(* CODESYS project EAS_PLC.library
   Company: ESCARRE AUTOMATIZACION Y SERVICIOS sl
   DefaultNamespace: EAS
   Version: 1.0.2
   Placeholder: EAS
   Author: EAS
   Title: EAS PLC

Project tree, tasks and I/O mapping:
  libraries: Tc2_Standard, * (Beckhoff Automation GmbH); Tc2_System, * (Beckhoff Automation GmbH); Tc3_Module, * (Beckhoff Automation GmbH); Util, * (System)
  DUTs/
    data type TipusCurva
  GVLs/
  POUs/
    PLC/
      MC/
        AddTanks/
          function block Circulation_TK [ST]
          function block fB_Intro_TK [ST]
          function block fBWash_TK [ST]
          function fCurvePerCen [ST]
        Elements/
          function block fBCalibrationLtr [ST]
          function block fBCntLiters [ST]
          function block fBHorn [ST]
          function block fbLiterCounter_by_flow [ST]
          function block fbLitersbyLevel [ST]
          function block fbMeterCounter_by_Speed [ST]
          function block fbPulseTrain [ST]
          function block fBUp_Down [ST]
          function block fbWashing_HT [ST]
        Fill/
          function block fBTemperatureFill [ST]
        Pump/
          function block fBPumpC [ST]
          function block fBPumpSpeed [ST]
        Seam/
          function block fBSeamTime [ST]
        Temperature/
          function block fBTermo [ST]
      Utils/
        AnalogConversions/
          function Canvi_Escala [ST]
          function Conv_Temp [ST]
        BitsConversions/
          function block Bits_to_Dword [ST]
          function block Bits_to_word [ST]
          function block Dword_to_bits [ST]
          function block Word_to_bits [ST]
        Counters/
          function block Calcul_Frequencia [ST]
          function block ContadorRapid [ST]
        FreqCycle/
          function block CalcFreq [ST]
          function block TCicle [ST]
        Timers/
          function block fBPulse1s [ST]
          function block TMP [ST]
          function block TMPpausa [ST]
  VISUs/
*)

// DUTs/TipusCurva
TYPE TipusCurva :
STRUCT
	Table:ARRAY [0..10] OF point;
END_STRUCT
END_TYPE

// POUs/PLC/MC/AddTanks/Circulation_TK
FUNCTION_BLOCK Circulation_TK
(*****************************************************************
Execute the recirculation of the add tank (Mac -> tank, tank -> mac) - 01/12/2021
v1.00
****************************************************************)
VAR_INPUT
	xActvRecirc:BOOL;				// Activate the function
	xPulsFinRecirc:BOOL;			// Finish the function
	xLowLevelRecirc:BOOL;			// Add tank Low level for the recirculation
	xHighLevelRecirc:BOOL;			// Add tank high level for the recirculation
	xMinimLevel:BOOL;				// Minimum tank level for the recirculation
	dwDrainTime:DWORD;				// Add tank drain time
END_VAR
VAR_OUTPUT
	xFiRecirc:BOOL;					// Recirculate finished
	xFill:BOOL;						// Add tank fill (runback)
	xIntro:BOOL;					// Add tank introduction (transfer)
END_VAR
VAR
	PararRecirculacio: BOOL;
	PararOmplerta: BOOL;
	OmplirEnRecirculacio: BOOL;
	PararIntroducio: BOOL;
	IntroduccioEnRecirculacio: BOOL;
	srPararRecirculacio : SR;
	TempoDescubrirNivBaix: TMP;
	Reircular: BOOL;
	FiBuidatCubeta: BOOL;
	BuidarCubeta: BOOL;
	TEmpoDrenatBuidat: TMP;
	srFiBuidatCubeta : SR;
END_VAR

// *********** Fin recircula por pulsador *****************
srPararRecirculacio(SET1:=xActvRecirc AND  xPulsFinRecirc, RESET:=NOT xActvRecirc , Q1=>PararRecirculacio );

Reircular := xActvRecirc AND NOT PararRecirculacio;

OmplirEnRecirculacio := Reircular AND NOT PararOmplerta;

IntroduccioEnRecirculacio := Reircular AND NOT PararIntroducio;
// ********* Pausa la introduccion si el nivel esta bajo *****************
TempoDescubrirNivBaix(xIN:=Reircular AND xLowLevelRecirc, dwSegons:=5 , xQ=> , dwTsegons=> );
PararIntroducio := NOT TempoDescubrirNivBaix.xQ; 

PararOmplerta := Reircular AND xHighLevelRecirc;

BuidarCubeta := xActvRecirc AND PararRecirculacio;

TEmpoDrenatBuidat(xIN:=BuidarCubeta AND NOT xMinimLevel, dwSegons:=dwDrainTime , xQ=> , dwTsegons=> );

srFiBuidatCubeta(SET1:=TEmpoDrenatBuidat.xQ , RESET:=NOT xActvRecirc , Q1=>FiBuidatCubeta );
// ************ Finaliza la recirculacion ********
xFiRecirc := FiBuidatCubeta;
// ************ Introduz a la maquina **********
xIntro := (BuidarCubeta AND NOT FiBuidatCubeta) OR IntroduccioEnRecirculacio;
// ************ Retorno de bano a la cubeta ********
xFill := OmplirEnRecirculacio;

END_FUNCTION_BLOCK

// POUs/PLC/Utils/Timers/TMP
FUNCTION_BLOCK TMP
(**********************************************************
Timer in seconds with a DWORD input - 29/11/2021
V1.0
*********************************************************)
VAR_INPUT
	xIN:BOOL;			// Enable Input
	dwSegons:DWORD;		// Setpoint Time (seconds) Input
END_VAR
VAR_OUTPUT
	xQ:BOOL;					// Boolean Output
	dwTsegons:DWORD;			// Currently Time (seconds) Output
END_VAR

VAR
	TEmporitz: TON;
	Temps: TIME;
	TempsTrans: TIME;
END_VAR

Temps := REAL_TO_TIME (DWORD_TO_REAL (dwSegons)*1000);

TEmporitz(IN:=xIN , PT:=Temps , Q=>xQ , ET=>TempsTrans );

dwTsegons := REAL_TO_DWORD(TIME_TO_REAL (TempsTrans)/1000);

END_FUNCTION_BLOCK

// POUs/PLC/MC/AddTanks/fB_Intro_TK
FUNCTION_BLOCK fB_Intro_TK
VAR_INPUT
	xActvIntro: BOOL;		///Enable the function
	dwCurve: DWORD;			/// Dosing curve
	dwTime: DWORD;			/// Duration Time
	rLevel: REAL;			/// Tank Level
	xLevelMin: BOOL;		/// Tank Minimun Level
	xIniCond: BOOL;			/// Initial condicions
	xPause: BOOL;			/// Pause the function
END_VAR
VAR_OUTPUT
	xFiIntro: BOOL;			/// End of the introduction
	rQTeoric: REAL;			/// Teoric Quantity of the introduction (%)
	rQreal: REAL;			/// Real Quantity of the introduction (%)
	xPrepareIntro: BOOL;	/// Prepare an Introduction
	xDosIntro: BOOL;		/// Introduct dosing (slow)
	xTransferIntro: BOOL;	/// Introduct transfering (fast)
	dwRemainingTime: DWORD;	/// Tiempo restante Intro
END_VAR
VAR
	IniciarIntro: BOOL;
	TEmpoInici: TMPPausa;
	calculQt: CHARCURVE;
	rampatems: RAMP_REAL;
	tempsreal: REAL;
	Tempsensegons: REAL;
	IntroduccioDosificada: BOOL;
	IntroduccioDirecte: BOOL;
	TempsEnPercentatge: REAL;
	TaulaCurva: ARRAY[0..10] OF point;
	RampaTempsInt: INT;
	QteoricaINT: INT;
	ERROR: BYTE;
	entradaRampa: REAL;
	NivellInicial: REAL;
	TempsNivellinim: TMPPausa;
	FiIntroDosificada: BOOL;
	TempsNivellinimDir: TMPPausa;
	FiDirecte: BOOL;
	srFiIntro: SR;
	A: INT;
	TMP_TimeRemaining: TMPPausa;
	dwActTime: DWORD;
END_VAR

// Inicia Intro
TEmpoInici(xIN:=xActvIntro AND xIniCond , dwSegons:=2 , xQ=>IniciarIntro , dwTsegons=> );

// Verifica si es introducion directa o dosificada
IF dwTime > 0
	THEN
		IntroduccioDosificada := TRUE;
		IntroduccioDirecte := FALSE;
	ELSE
		IntroduccioDosificada := FALSE;
		IntroduccioDirecte := TRUE;
END_IF

// Calculos del tiempo
Tempsensegons := DWORD_TO_REAL(dwTime*60);

IF IniciarIntro
	THEN
		EntradaRampa := Tempsensegons;
	ELSE
		EntradaRampa := 0;	
		NivellInicial := rLevel;
END_IF

// Si es introducin dosificada calcula la rampa
IF IntroduccioDosificada
	THEN
		rampatems(
			IN:= EntradaRampa, 
			ASCEND:= 1, 
			DESCEND:= Tempsensegons, 
			TIMEBASE:= T#1S, 
			RESET:= (IniciarIntro AND xPause) , 
			OUT=> tempsreal);

		TempsEnPercentatge := (tempsreal/Tempsensegons)*100;
END_IF

RampaTempsInt := REAL_TO_INT(TempsEnPercentatge*100);

TaulaCurva :=  fCurvePerCen(Curve:=DWORD_TO_INT (dwCurve));

calculQt(
	IN:= RampaTempsInt , 
	N:=11 , 
	P:=TaulaCurva , 
	OUT=>QteoricaINT , 
	ERR=>ERROR );

// Si se ha iniciado la introducion calcula el Qreal
IF IniciarIntro AND NivellInicial > 0
	THEN
		rQreal := (rLevel/NivellInicial)*100;
END_IF

rQTeoric := (INT_TO_REAL(QteoricaINT))/100;

xPrepareIntro := IniciarIntro AND NOT xFiIntro;

IF (rQreal > rQTeoric AND IniciarIntro AND IntroduccioDosificada AND NOT xFiIntro AND IniciarIntro) 
		THEN
		xDosIntro := TRUE;
	ELSE
		xDosIntro := FALSE;
END_IF

xTransferIntro := NOT(IntroduccioDosificada) AND IniciarIntro AND NOT xFiIntro;

TempsNivellinim(xIN:=NOT(xLevelMin) , dwSegons:=60 , xQ=> , dwTsegons=> );

IF 	rQTeoric <= 0 OR 
	rQTeoric <= 0 OR 
	TempsNivellinim.xQ (* OR 
	IntroduccioDosificada OR 
	IniciarIntro OR 
	NOT xLevelMin *)
	THEN
		FiIntroDosificada := TRUE;
	ELSE
		FiIntroDosificada := FALSE;
END_IF

TempsNivellinimDir(xIN:= NOT xLevelMin , dwSegons:=3 , xQ=> , dwTsegons=> );

FiDirecte := NOT IntroduccioDosificada AND IniciarIntro AND TempsNivellinimDir.xQ;


srFiIntro(  SET1:=(FiIntroDosificada OR FiDirecte) AND xActvIntro, 
			RESET:= NOT xActvIntro , Q1=>xFiIntro);

// TIEMPO RESTANTE INTRO
TMP_TimeRemaining(
	xIN:= IniciarIntro , 
	xPausa:= xPause, 
	dwSegons:= (dwTime*60), 
	xQ=> , 
	dwTsegons=> dwActTime, 
	rTsegons=> );

dwRemainingTime:= (dwTime*60)- dwActTime;


A:=A+1;

END_FUNCTION_BLOCK

// POUs/PLC/MC/AddTanks/fCurvePerCen
FUNCTION fCurvePerCen : ARRAY [0..10] OF POINT
(*******************************************************
Aquest Bloc Carrega per HardCode els valors de les les Corves percentuals.
Al demanar una corva retorna una taula de punts per a l'introduccio
=========================================
06/09/2006= Error corva7.
********************************************************)
VAR_INPUT
	Curve:INT;			// Curve (0 - 19)
END_VAR

VAR_OUTPUT

END_VAR	

VAR
END_VAR



(*Curve 0*)
IF Curve=0 THEN
fCurvePerCen[0].X:=0;
fCurvePerCen[0].Y:=10000;
fCurvePerCen[1].X:=1000;
fCurvePerCen[1].Y:=9000;
fCurvePerCen[2].X:=2000;
fCurvePerCen[2].Y:=8000;
fCurvePerCen[3].X:=3000;
fCurvePerCen[3].Y:=7000;
fCurvePerCen[4].X:=4000;
fCurvePerCen[4].Y:=6000;
fCurvePerCen[5].X:=5000;
fCurvePerCen[5].Y:=5000;
fCurvePerCen[6].X:=6000;
fCurvePerCen[6].Y:=4000;
fCurvePerCen[7].X:=7000;
fCurvePerCen[7].Y:=3000;
fCurvePerCen[8].X:=8000;
fCurvePerCen[8].Y:=2000;
fCurvePerCen[9].X:=9000;
fCurvePerCen[9].Y:=1000;
fCurvePerCen[10].X:=10000;
fCurvePerCen[10].Y:=0;
END_IF


(*Curve 1*)
IF curve=1 THEN
	fCurvePerCen[0].X:=0;
	fCurvePerCen[0].Y:=10000;
	fCurvePerCen[1].X:=1000;
	fCurvePerCen[1].Y:=9100;
	fCurvePerCen[2].X:=2000;
	fCurvePerCen[2].Y:=8200;
	fCurvePerCen[3].X:=3000;
	fCurvePerCen[3].Y:=7300;
	fCurvePerCen[4].X:=4000;
	fCurvePerCen[4].Y:=6400;
	fCurvePerCen[5].X:=5000;
	fCurvePerCen[5].Y:=5400;
	fCurvePerCen[6].X:=6000;
	fCurvePerCen[6].Y:=4500;
	fCurvePerCen[7].X:=7000;
	fCurvePerCen[7].Y:=3500;
	fCurvePerCen[8].X:=8000;
	fCurvePerCen[8].Y:=2400;
	fCurvePerCen[9].X:=9000;
	fCurvePerCen[9].Y:=1300;
	fCurvePerCen[10].X:=10000;
	fCurvePerCen[10].Y:=0;
END_IF


(*Curve 2*)
IF curve=2 THEN
	fCurvePerCen[0].X:=0;
	fCurvePerCen[0].Y:=10000;
	fCurvePerCen[1].X:=1000;
	fCurvePerCen[1].Y:=9200;
	fCurvePerCen[2].X:=2000;
	fCurvePerCen[2].Y:=8400;
	fCurvePerCen[3].X:=3000;
	fCurvePerCen[3].Y:=7600;
	fCurvePerCen[4].X:=4000;
	fCurvePerCen[4].Y:=6700;
	fCurvePerCen[5].X:=5000;
	fCurvePerCen[5].Y:=5800;
	fCurvePerCen[6].X:=6000;
	fCurvePerCen[6].Y:=4900;
	fCurvePerCen[7].X:=7000;
	fCurvePerCen[7].Y:=3900;
	fCurvePerCen[8].X:=8000;
	fCurvePerCen[8].Y:=2800;
	fCurvePerCen[9].X:=9000;
	fCurvePerCen[9].Y:=1500;
	fCurvePerCen[10].X:=10000;
	fCurvePerCen[10].Y:=0;
END_IF

(*GVL.Curve 3*)
IF Curve=3 THEN
	fCurvePerCen[0].X:=0;
	fCurvePerCen[0].Y:=10000;
	fCurvePerCen[1].X:=1000;
	fCurvePerCen[1].Y:=9300;
	fCurvePerCen[2].X:=2000;
	fCurvePerCen[2].Y:=8500;
	fCurvePerCen[3].X:=3000;
	fCurvePerCen[3].Y:=7800;
	fCurvePerCen[4].X:=4000;
	fCurvePerCen[4].Y:=7000;
	fCurvePerCen[5].X:=5000;
	fCurvePerCen[5].Y:=6200;
	fCurvePerCen[6].X:=6000;
	fCurvePerCen[6].Y:=5300;
	fCurvePerCen[7].X:=7000;
	fCurvePerCen[7].Y:=4400;
	fCurvePerCen[8].X:=8000;
	fCurvePerCen[8].Y:=3200;
	fCurvePerCen[9].X:=9000;
	fCurvePerCen[9].Y:=1800;
	fCurvePerCen[10].X:=10000;
	fCurvePerCen[10].Y:=0;
END_IF

(*GVL.Curve 4*)
IF curve=4 THEN
	fCurvePerCen[0].X:=0;
	fCurvePerCen[0].Y:=10000;
	fCurvePerCen[1].X:=1000;
	fCurvePerCen[1].Y:=9400;
	fCurvePerCen[2].X:=2000;
	fCurvePerCen[2].Y:=8600;
	fCurvePerCen[3].X:=3000;
	fCurvePerCen[3].Y:=8100;
	fCurvePerCen[4].X:=4000;
	fCurvePerCen[4].Y:=7400;
	fCurvePerCen[5].X:=5000;
	fCurvePerCen[5].Y:=6600;
	fCurvePerCen[6].X:=6000;
	fCurvePerCen[6].Y:=5700;
	fCurvePerCen[7].X:=7000;
	fCurvePerCen[7].Y:=4900;
	fCurvePerCen[8].X:=8000;
	fCurvePerCen[8].Y:=3600;
	fCurvePerCen[9].X:=9000;
	fCurvePerCen[9].Y:=2100;
	fCurvePerCen[10].X:=10000;
	fCurvePerCen[10].Y:=0;
END_IF


(*GVL.Curve 5*)
IF curve=5 THEN
	fCurvePerCen[0].X:=0;
	fCurvePerCen[0].Y:=10000;
	fCurvePerCen[1].X:=1000;
	fCurvePerCen[1].Y:=9500;
	fCurvePerCen[2].X:=2000;
	fCurvePerCen[2].Y:=8800;
	fCurvePerCen[3].X:=3000;
	fCurvePerCen[3].Y:=8300;
	fCurvePerCen[4].X:=4000;
	fCurvePerCen[4].Y:=7600;
	fCurvePerCen[5].X:=5000;
	fCurvePerCen[5].Y:=7000;
	fCurvePerCen[6].X:=6000;
	fCurvePerCen[6].Y:=6200;
	fCurvePerCen[7].X:=7000;
	fCurvePerCen[7].Y:=5400;
	fCurvePerCen[8].X:=8000;
	fCurvePerCen[8].Y:=4000;
	fCurvePerCen[9].X:=9000;
	fCurvePerCen[9].Y:=2300;
	fCurvePerCen[10].X:=10000;
	fCurvePerCen[10].Y:=0;
END_IF


(*GVL.Curve 6*)
IF curve=6 THEN
	fCurvePerCen[0].X:=0;
	fCurvePerCen[0].Y:=10000;
	fCurvePerCen[1].X:=1000;
	fCurvePerCen[1].Y:=9500;
	fCurvePerCen[2].X:=2000;
	fCurvePerCen[2].Y:=9000;
	fCurvePerCen[3].X:=3000;
	fCurvePerCen[3].Y:=8500;
	fCurvePerCen[4].X:=4000;
	fCurvePerCen[4].Y:=8000;
	fCurvePerCen[5].X:=5000;
	fCurvePerCen[5].Y:=7400;
	fCurvePerCen[6].X:=6000;
	fCurvePerCen[6].Y:=6600;
	fCurvePerCen[7].X:=7000;
	fCurvePerCen[7].Y:=5800;
	fCurvePerCen[8].X:=8000;
	fCurvePerCen[8].Y:=4400;
	fCurvePerCen[9].X:=9000;
	fCurvePerCen[9].Y:=2600;
	fCurvePerCen[10].X:=10000;
	fCurvePerCen[10].Y:=0;
END_IF


(*GVL.Curve 7*)
IF curve=7 THEN
	fCurvePerCen[0].X:=0;
	fCurvePerCen[0].Y:=10000;
	fCurvePerCen[1].X:=1000;
	fCurvePerCen[1].Y:=9600;
	fCurvePerCen[2].X:=2000;
	fCurvePerCen[2].Y:=9200;
	fCurvePerCen[3].X:=3000;
	fCurvePerCen[3].Y:=8800;
	fCurvePerCen[4].X:=4000;
	fCurvePerCen[4].Y:=8300;
	fCurvePerCen[5].X:=5000;
	fCurvePerCen[5].Y:=7800;
	fCurvePerCen[6].X:=6000;
	fCurvePerCen[6].Y:=7100;
	fCurvePerCen[7].X:=7000;
	fCurvePerCen[7].Y:=6300;
	fCurvePerCen[8].X:=8000;
	fCurvePerCen[8].Y:=4800;
	fCurvePerCen[9].X:=9000;
	fCurvePerCen[9].Y:=2800;
	fCurvePerCen[10].X:=10000;
	fCurvePerCen[10].Y:=0;
END_IF


(*GVL.Curve 8*)
IF curve=8 THEN
	fCurvePerCen[0].X:=0;
	fCurvePerCen[0].Y:=10000;
	fCurvePerCen[1].X:=1000;
	fCurvePerCen[1].Y:=9700;
	fCurvePerCen[2].X:=2000;
	fCurvePerCen[2].Y:=9400;
	fCurvePerCen[3].X:=3000;
	fCurvePerCen[3].Y:=9100;
	fCurvePerCen[4].X:=4000;
	fCurvePerCen[4].Y:=8600;
	fCurvePerCen[5].X:=5000;
	fCurvePerCen[5].Y:=8200;
	fCurvePerCen[6].X:=6000;
	fCurvePerCen[6].Y:=7500;
	fCurvePerCen[7].X:=7000;
	fCurvePerCen[7].Y:=6700;
	fCurvePerCen[8].X:=8000;
	fCurvePerCen[8].Y:=5200;
	fCurvePerCen[9].X:=9000;
	fCurvePerCen[9].Y:=3100;
	fCurvePerCen[10].X:=10000;
	fCurvePerCen[10].Y:=0;
END_IF

(*GVL.Curve 9*)
IF curve=9 THEN
	fCurvePerCen[0].X:=0;
	fCurvePerCen[0].Y:=10000;
	fCurvePerCen[1].X:=1000;
	fCurvePerCen[1].Y:=9800;
	fCurvePerCen[2].X:=2000;
	fCurvePerCen[2].Y:=9600;
	fCurvePerCen[3].X:=3000;
	fCurvePerCen[3].Y:=9300;
	fCurvePerCen[4].X:=4000;
	fCurvePerCen[4].Y:=9000;
	fCurvePerCen[5].X:=5000;
	fCurvePerCen[5].Y:=8600;
	fCurvePerCen[6].X:=6000;
	fCurvePerCen[6].Y:=7900;
	fCurvePerCen[7].X:=7000;
	fCurvePerCen[7].Y:=7100;
	fCurvePerCen[8].X:=8000;
	fCurvePerCen[8].Y:=5600;
	fCurvePerCen[9].X:=9000;
	fCurvePerCen[9].Y:=3400;
	fCurvePerCen[10].X:=10000;
	fCurvePerCen[10].Y:=0;
END_IF 

(*GVL.Curve 10*)
IF curve=10 THEN
	fCurvePerCen[0].X:=0;
	fCurvePerCen[0].Y:=10000;
	fCurvePerCen[1].X:=1000;
	fCurvePerCen[1].Y:=9000;
	fCurvePerCen[2].X:=2000;
	fCurvePerCen[2].Y:=8000;
	fCurvePerCen[3].X:=3000;
	fCurvePerCen[3].Y:=7000;
	fCurvePerCen[4].X:=4000;
	fCurvePerCen[4].Y:=6000;
	fCurvePerCen[5].X:=5000;
	fCurvePerCen[5].Y:=5000;
	fCurvePerCen[6].X:=6000;
	fCurvePerCen[6].Y:=4000;
	fCurvePerCen[7].X:=7000;
	fCurvePerCen[7].Y:=3000;
	fCurvePerCen[8].X:=8000;
	fCurvePerCen[8].Y:=2000;
	fCurvePerCen[9].X:=9000;
	fCurvePerCen[9].Y:=1000;
	fCurvePerCen[10].X:=10000;
	fCurvePerCen[10].Y:=0;
END_IF
	
	
(*GVL.Curve 11*)
IF curve=11 THEN
	fCurvePerCen[0].X:=0;
	fCurvePerCen[0].Y:=10000;
	fCurvePerCen[1].X:=1000;
	fCurvePerCen[1].Y:=8700;
	fCurvePerCen[2].X:=2000;
	fCurvePerCen[2].Y:=7600;
	fCurvePerCen[3].X:=3000;
	fCurvePerCen[3].Y:=6500;
	fCurvePerCen[4].X:=4000;
	fCurvePerCen[4].Y:=5500;
	fCurvePerCen[5].X:=5000;
	fCurvePerCen[5].Y:=4600;
	fCurvePerCen[6].X:=6000;
	fCurvePerCen[6].Y:=3600;
	fCurvePerCen[7].X:=7000;
	fCurvePerCen[7].Y:=2700;
	fCurvePerCen[8].X:=8000;
	fCurvePerCen[8].Y:=1800;
	fCurvePerCen[9].X:=9000;
	fCurvePerCen[9].Y:=900;
	fCurvePerCen[10].X:=10000;
	fCurvePerCen[10].Y:=0;
END_IF


(*GVL.Curve 12*)
IF curve=12 THEN
	fCurvePerCen[0].X:=0;
	fCurvePerCen[0].Y:=10000;
	fCurvePerCen[1].X:=1000;
	fCurvePerCen[1].Y:=8500;
	fCurvePerCen[2].X:=2000;
	fCurvePerCen[2].Y:=7200;
	fCurvePerCen[3].X:=3000;
	fCurvePerCen[3].Y:=6100;
	fCurvePerCen[4].X:=4000;
	fCurvePerCen[4].Y:=5100;
	fCurvePerCen[5].X:=5000;
	fCurvePerCen[5].Y:=4200;
	fCurvePerCen[6].X:=6000;
	fCurvePerCen[6].Y:=3300;
	fCurvePerCen[7].X:=7000;
	fCurvePerCen[7].Y:=2400;
	fCurvePerCen[8].X:=8000;
	fCurvePerCen[8].Y:=1600;
	fCurvePerCen[9].X:=9000;
	fCurvePerCen[9].Y:=800;
	fCurvePerCen[10].X:=10000;
	fCurvePerCen[10].Y:=0;
END_IF


(*GVL.Curve 13*)
IF curve=13 THEN
	fCurvePerCen[0].X:=0;
	fCurvePerCen[0].Y:=10000;
	fCurvePerCen[1].X:=1000;
	fCurvePerCen[1].Y:=8200;
	fCurvePerCen[2].X:=2000;
	fCurvePerCen[2].Y:=6800;
	fCurvePerCen[3].X:=3000;
	fCurvePerCen[3].Y:=5600;
	fCurvePerCen[4].X:=4000;
	fCurvePerCen[4].Y:=4700;
	fCurvePerCen[5].X:=5000;
	fCurvePerCen[5].Y:=3800;
	fCurvePerCen[6].X:=6000;
	fCurvePerCen[6].Y:=3000;
	fCurvePerCen[7].X:=7000;
	fCurvePerCen[7].Y:=2200;
	fCurvePerCen[8].X:=8000;
	fCurvePerCen[8].Y:=1500;
	fCurvePerCen[9].X:=9000;
	fCurvePerCen[9].Y:=700;
	fCurvePerCen[10].X:=10000;
	fCurvePerCen[10].Y:=0;
END_IF


(*GVL.Curve 14*)
IF curve=14 THEN
	fCurvePerCen[0].X:=0;
	fCurvePerCen[0].Y:=10000;
	fCurvePerCen[1].X:=1000;
	fCurvePerCen[1].Y:=7900;
	fCurvePerCen[2].X:=2000;
	fCurvePerCen[2].Y:=6400;
	fCurvePerCen[3].X:=3000;
	fCurvePerCen[3].Y:=5100;
	fCurvePerCen[4].X:=4000;
	fCurvePerCen[4].Y:=4300;
	fCurvePerCen[5].X:=5000;
	fCurvePerCen[5].Y:=3400;
	fCurvePerCen[6].X:=6000;
	fCurvePerCen[6].Y:=2600;
	fCurvePerCen[7].X:=5000;
	fCurvePerCen[7].Y:=1900;
	fCurvePerCen[8].X:=8000;
	fCurvePerCen[8].Y:=1400;
	fCurvePerCen[9].X:=9000;
	fCurvePerCen[9].Y:=600;
	fCurvePerCen[10].X:=10000;
	fCurvePerCen[10].Y:=0;
END_IF


(*GVL.Curve 15*)
IF curve=15 THEN
	fCurvePerCen[0].X:=0;
	fCurvePerCen[0].Y:=10000;
	fCurvePerCen[1].X:=1000;
	fCurvePerCen[1].Y:=7700;
	fCurvePerCen[2].X:=2000;
	fCurvePerCen[2].Y:=6000;
	fCurvePerCen[3].X:=3000;
	fCurvePerCen[3].Y:=4600;
	fCurvePerCen[4].X:=4000;
	fCurvePerCen[4].Y:=3800;
	fCurvePerCen[5].X:=5000;
	fCurvePerCen[5].Y:=3000;
	fCurvePerCen[6].X:=6000;
	fCurvePerCen[6].Y:=2400;
	fCurvePerCen[7].X:=7000;
	fCurvePerCen[7].Y:=1700;
	fCurvePerCen[8].X:=8000;
	fCurvePerCen[8].Y:=1200;
	fCurvePerCen[9].X:=9000;
	fCurvePerCen[9].Y:=500;
	fCurvePerCen[10].X:=10000;
	fCurvePerCen[10].Y:=0;
END_IF

(*GVL.Curve 16*)
IF curve=16 THEN
	fCurvePerCen[0].X:=0;
	fCurvePerCen[0].Y:=10000;
	fCurvePerCen[1].X:=1000;
	fCurvePerCen[1].Y:=7400;
	fCurvePerCen[2].X:=2000;
	fCurvePerCen[2].Y:=5600;
	fCurvePerCen[3].X:=3000;
	fCurvePerCen[3].Y:=4200;
	fCurvePerCen[4].X:=4000;
	fCurvePerCen[4].Y:=3400;
	fCurvePerCen[5].X:=5000;
	fCurvePerCen[5].Y:=2600;
	fCurvePerCen[6].X:=6000;
	fCurvePerCen[6].Y:=2000;
	fCurvePerCen[7].X:=7000;
	fCurvePerCen[7].Y:=1500;
	fCurvePerCen[8].X:=8000;
	fCurvePerCen[8].Y:=1000;
	fCurvePerCen[9].X:=9000;
	fCurvePerCen[9].Y:=500;
	fCurvePerCen[10].X:=10000;
	fCurvePerCen[10].Y:=0;
END_IF


(*GVL.Curve 17*)
IF curve=17 THEN
	fCurvePerCen[0].X:=0;
	fCurvePerCen[0].Y:=10000;
	fCurvePerCen[1].X:=1000;
	fCurvePerCen[1].Y:=7200;
	fCurvePerCen[2].X:=2000;
	fCurvePerCen[2].Y:=5200;
	fCurvePerCen[3].X:=3000;
	fCurvePerCen[3].Y:=3700;
	fCurvePerCen[4].X:=4000;
	fCurvePerCen[4].Y:=2900;
	fCurvePerCen[5].X:=5000;
	fCurvePerCen[5].Y:=2200;
	fCurvePerCen[6].X:=6000;
	fCurvePerCen[6].Y:=1700;
	fCurvePerCen[7].X:=7000;
	fCurvePerCen[7].Y:=1200;
	fCurvePerCen[8].X:=8000;
	fCurvePerCen[8].Y:=800;
	fCurvePerCen[9].X:=9000;
	fCurvePerCen[9].Y:=400;
	fCurvePerCen[10].X:=10000;
	fCurvePerCen[10].Y:=0;
END_IF


(*GVL.Curve 18*)
IF curve=18 THEN
	fCurvePerCen[0].X:=0;
	fCurvePerCen[0].Y:=10000;
	fCurvePerCen[1].X:=1000;
	fCurvePerCen[1].Y:=6900;
	fCurvePerCen[2].X:=2000;
	fCurvePerCen[2].Y:=4800;
	fCurvePerCen[3].X:=3000;
	fCurvePerCen[3].Y:=3300;
	fCurvePerCen[4].X:=4000;
	fCurvePerCen[4].Y:=2500;
	fCurvePerCen[5].X:=5000;
	fCurvePerCen[5].Y:=1800;
	fCurvePerCen[6].X:=6000;
	fCurvePerCen[6].Y:=1400;
	fCurvePerCen[7].X:=7000;
	fCurvePerCen[7].Y:=900;
	fCurvePerCen[8].X:=8000;
	fCurvePerCen[8].Y:=600;
	fCurvePerCen[9].X:=9000;
	fCurvePerCen[9].Y:=300;
	fCurvePerCen[10].X:=10000;
	fCurvePerCen[10].Y:=0;
END_IF


(*GVL.Curve 19*)
IF curve=19 THEN
	fCurvePerCen[0].X:=0;
	fCurvePerCen[0].Y:=10000;
	fCurvePerCen[1].X:=1000;
	fCurvePerCen[1].Y:=6600;
	fCurvePerCen[2].X:=2000;
	fCurvePerCen[2].Y:=4400;
	fCurvePerCen[3].X:=3000;
	fCurvePerCen[3].Y:=2900;
	fCurvePerCen[4].X:=4000;
	fCurvePerCen[4].Y:=1900;
	fCurvePerCen[5].X:=5000;
	fCurvePerCen[5].Y:=1400;
	fCurvePerCen[6].X:=6000;
	fCurvePerCen[6].Y:=1000;
	fCurvePerCen[7].X:=7000;
	fCurvePerCen[7].Y:=700;
	fCurvePerCen[8].X:=8000;
	fCurvePerCen[8].Y:=400;
	fCurvePerCen[9].X:=9000;
	fCurvePerCen[9].Y:=200;
	fCurvePerCen[10].X:=10000;
	fCurvePerCen[10].Y:=0;
END_IF

END_FUNCTION

// POUs/PLC/Utils/Timers/TMPpausa
FUNCTION_BLOCK TMPpausa
(**********************************************************
Timer in seconds (DWORD input) and an pause Input - 29/11/2021
V1.0
*********************************************************)
VAR_INPUT
	xIN:BOOL;				// Enable Input
	xPausa:BOOL;			// Pause Input
	dwSegons:DWORD;			// Setpoint Time in seconds (DWORD)
END_VAR
VAR_OUTPUT					
	xQ:BOOL;				// Boolean Output
	dwTsegons:DWORD;		// ET time in seconds(DWORD)
	rTsegons: REAL;			// ET time in seconds(REAL)

END_VAR

VAR
	TEmporitz: TON;
	Temps: TIME;
	TempsTrans: TIME;
	Pols_fin: F_TRIG;
	reset: BOOL;
	Temps_contador: TIME;
	Temps_pausa: TIME;
	contgeActual: TIME;
END_VAR

Temps := REAL_TO_TIME (DWORD_TO_REAL (dwSegons)*1000);

Pols_fin(CLK:=xPausa , Q=>reset);

IF	xPausa 
	THEN
		contgeActual := TEmporitz.ET;
END_IF

IF xPausa AND contgeActual > T#0S
	THEN
		Temps_pausa:= contgeActual;
		TempsTrans := Temps_pausa + TempsTrans; 
END_IF

TEmps_contador := Temps-TempsTrans;

TEmporitz(IN:=xIn AND NOT xPausa AND NOT reset, PT:=TEmps_contador , Q=>xQ , ET=>contgeActual );

IF NOT xIn
	THEN
	TEmps_contador := t#0s;
	TempsTrans := t#0s;
	Temps_pausa:= t#0s;
END_IF

dwTsegons := (REAL_TO_DWORD(TIME_TO_REAL((contgeActual)+(TempsTrans)))/1000);
rTsegons := ((TIME_TO_REAL((contgeActual)+(TempsTrans)))/1000);

END_FUNCTION_BLOCK

// POUs/PLC/MC/AddTanks/fBWash_TK
FUNCTION_BLOCK fBWash_TK
VAR_INPUT
	/// Enable function input
	xStartWash: BOOL;
	/// Minimum Level Input
	xMinimLevel: BOOL;
	/// Delay to detect the low level
	dwDetectLowLevelTime: DWORD;
	/// Drain Time
	dwDrainTime: DWORD;
	/// 1st Wash Time
	dw1stWashTime: DWORD;
	/// 2nd Wash Time
	dw2ndWashTime: DWORD;
	/// 3rd Wash Time
	dw3rdWashTime: DWORD;
	/// Drain Option (0 - 3)
	DrainType: DWORD;
END_VAR
VAR_OUTPUT
	/// Function finished			
	xFinWash: BOOL;
	/// Fill the add tank output
	xWash: BOOL;
	/// Transfer add tank to machine
	xToMachine: BOOL;
	/// Drain add tank
	xToDrain: BOOL;
END_VAR
VAR
	FerTotsElsRentats: BOOL;
	NomesRentatsAMaquina: BOOL;
	NoFerRentats: BOOL;
	FiPrimerRentat: BOOL;
	PrimerRentat: BOOL;
	TempoPrimerRentat: TMPPausa;
	FiPrimerBuidat: BOOL;
	PrimerBuidat: BOOL;
	FiSegonRentat: BOOL;
	SegonRentat: BOOL;
	FiSegonBuidat: BOOL;
	SegonBuidat: BOOL;
	TempoPrimerBuidat: TMPPausa;
	TempoSegonRentat: TMPPausa;
	TempoSegonBuidat: TMPPausa;
	TempoTercerRentat: TMPPausa;
	TempoTercerBuidat: TMPPausa;
	FiTercerRentat: BOOL;
	TercerRentat: BOOL;
	FiTercerBuidat: BOOL;
	TercerBuidat: BOOL;
	TempoBuit: TON;
	ComencaArentar: BOOL;
	BuidaDelTot: BOOL;
	srComencaArentar: SR;
	srFiPrimerRentat: SR;
	srFiPrimerBuidat: SR;
	srFiSegonRentat: SR;
	srFiSegonBuidat: SR;
	srFiTercerRentat: SR;
	srFiTercerBuidat: SR;
	FiTercer: BOOL;
	D: TMPPausa;
END_VAR

// ********** Define el tipo de lavado ***********
CASE DrainType OF
	0 : FerTotsElsRentats := TRUE;
		NoFerRentats := FALSE;
		NomesRentatsAMaquina := FALSE;
	1 : FerTotsElsRentats := FALSE;
		NoFerRentats := TRUE;
		NomesRentatsAMaquina := FALSE;
	2 : FerTotsElsRentats := FALSE;
		NoFerRentats := FALSE;
		NomesRentatsAMaquina := TRUE;
	3 : FerTotsElsRentats := TRUE;
		NoFerRentats := FALSE;
		NomesRentatsAMaquina := FALSE;
END_CASE

// ************** Empeza el lavado **************
TempoBuit(IN:= xStartWash AND NOT xMinimLevel, PT:=T#2S , Q=> , ET=> );

srComencaArentar(SET1:=TempoBuit.Q , RESET:= NOT xStartWash , Q1=>ComencaArentar );

BuidaDelTot := xStartWash AND NOT ComencaArentar;

// ********** Control Primer Lavado ******************
PrimerRentat := ComencaArentar AND NOT FiPrimerRentat;

TempoPrimerRentat(
	xIN:= ComencaArentar, 
	xPausa:= , 
	dwSegons:= dw1stWashTime, 
	xQ=> , 
	dwTsegons=> , 
	rTsegons=> );

srFiPrimerRentat(SET1:=TempoPrimerRentat.XQ , RESET:= NOT xStartWash , Q1=>FiPrimerRentat );

PrimerBuidat := FiPrimerRentat AND NOT FiPrimerBuidat;

TempoPrimerBuidat(
	xIN:= PrimerBuidat AND NOT  xMinimLevel, 
	xPausa:= , 
	dwSegons:=dwDetectLowLevelTime , 
	xQ=> , 
	dwTsegons=> , 
	rTsegons=> );

srFiPrimerBuidat(SET1:=TempoPrimerBuidat.XQ , RESET:=NOT xStartWash  , Q1=>FiPrimerBuidat );



// ********** Control Segun Lavado ***************** 
SegonRentat := FiPrimerBuidat AND NOT FiSegonRentat;

TempoSegonRentat(
	xIN:= SegonRentat , 
	xPausa:= , 
	dwSegons:= dw2ndWashTime, 
	xQ=> , 
	dwTsegons=> , 
	rTsegons=> );

srFiSegonRentat(SET1:=TempoSegonRentat.XQ , RESET:=NOT xStartWash  , Q1=>FiSegonRentat );

SegonBuidat := FiSegonRentat AND NOT FiSegonBuidat;

TempoSegonBuidat(
	xIN:= SegonBuidat AND NOT xMinimLevel, 
	xPausa:= , 
	dwSegons:= dwDetectLowLevelTime, 
	xQ=> , 
	dwTsegons=> , 
	rTsegons=> );

srFiSegonBuidat(SET1:=TempoSegonBuidat.XQ , RESET:=NOT xStartWash  , Q1=>FiSegonBuidat );

// ********** Control Tercer Lavado ***************** 
TercerRentat := FiSegonBuidat AND NOT FiTercerRentat;

TempoTercerRentat(
	xIN:= TercerRentat, 
	xPausa:= , 
	dwSegons:= dw3rdWashTime, 
	xQ=> , 
	dwTsegons=> , 
	rTsegons=> );

srFiTercerRentat(SET1:=TempoTercerRentat.XQ , RESET:=NOT xStartWash  , Q1=>FiTercerRentat );

TercerBuidat := FiTercerRentat AND NOT FiTercerBuidat;

TempoTercerBuidat(
	xIN:= TercerBuidat AND NOT xMinimLevel, 
	xPausa:= , 
	dwSegons:= dwDrainTime, 
	xQ=> , 
	dwTsegons=> , 
	rTsegons=> );

srFiTercerBuidat(SET1:=TempoTercerBuidat.XQ , RESET:=NOT xStartWash  , Q1=>FiTercerBuidat);

// ************* Finaliza los lavados ****************
xFinWash := xStartWash AND ((FerTotsElsRentats AND FiTercerBuidat) OR 
							(NomesRentatsAMaquina AND FiSegonBuidat) OR 
							NoFerRentats);// AND FiPrimerBuidat));

IF xFinWash THEN
	xStartWash := FALSE;
END_IF

// ************** Activa salidas *************
xWash	:= xStartWash AND (PrimerRentat OR SegonRentat OR TercerRentat);

xToMachine := NOT xFinWash AND (PrimerBuidat OR SegonBuidat OR BuidaDelTot);

xToDrain := NOT xFinWash AND TercerBuidat;

END_FUNCTION_BLOCK

// POUs/PLC/MC/Elements/fBCalibrationLtr
FUNCTION_BLOCK fBCalibrationLtr
//*************************************************************************************
// Con esta funcion se calibra el factor de forma de 
//
//
//*************************************************************************************

VAR_INPUT
	xStart: BOOL;		///Inicio Calibracion
	xSegOK: BOOL;		///Seguridades de máquina ok (Temp. block o Presión Min.)
	wNivel: WORD;		///Analógica de nivel debe estar ser entre 0 y 100%
	rLitros: REAL;		///Valor de litros en real
	xPause: BOOL;		///Pausa la calibracion cerrando el agua de entrada
END_VAR
VAR_OUTPUT
	N00: WORD;
	N10: WORD;
	N20: WORD;
	N30: WORD;
	N40: WORD;
	N50: WORD;
	N60: WORD;
	N70: WORD;
	N80: WORD;
	N90: WORD;
	N100: WORD;

	xPolsResetCntLitros: BOOL; 	///Usarlo para resetear el cuentalitros al inicio
	xLlenado: BOOL;				///Salida de llenado de maquina
	xAlMacNoVacia: BOOL;		///Alarma maquina no vacia al inicio.
	xFinCalibracion: BOOL;		///Pulso Fin Calibracion 2 seg
	rLitrosNivel: REAL;			///Litros extraidos del nivel
END_VAR

VAR
	xAMcNoVacia: BOOL;
	xInicioCalibracion: BOOL;
	RS_InicioCalibracion: RS;
	TON_FinCal: TON;
	TP_ResetCuentalitros: TP;
	TP_FinCalibracion: TP;
END_VAR


//Verificar que nivel es 0 antes de calibrar
xAMcNoVacia:= xStart AND NOT (xInicioCalibracion) AND (wNivel>=1);

// Inicio Calibracion
RS_InicioCalibracion(SET:= xStart AND (wNivel<=1), RESET1:= NOT (xStart)OR TON_FinCal.Q, Q1=> );
xInicioCalibracion:= RS_InicioCalibracion.Q1;

// Pulso al inicio para resetear el cuentalitros
TP_ResetCuentalitros(IN:= xInicioCalibracion, PT:= T#1S, Q=> , ET=> );
xPolsResetCntLitros:=TP_ResetCuentalitros.Q;

//Resetear los valores anteriores al iniciar Calibrado
IF xPolsResetCntLitros
	THEN
	N00 := 0;
	N10 := 0;
	N20 := 0;
	N30 := 0;
	N40 := 0;
	N50 := 0;
	N60 := 0;
	N70 := 0;
	N80 := 0;
	N90 := 0;
	N100 := 0;
END_IF

//Calibracion de la máquina
IF xInicioCalibracion THEN
	CASE wNivel OF
					
		0:	
			N00 := REAL_TO_WORD (rLitros);
		10:	
			N10 := REAL_TO_WORD (rLitros);
		20:	
			N20 := REAL_TO_WORD (rLitros);
		30:	
			N30 := REAL_TO_WORD (rLitros);
		40:	
			N40 := REAL_TO_WORD (rLitros);
		50:	
			N50 := REAL_TO_WORD (rLitros);
		60:	
			N60 := REAL_TO_WORD (rLitros);
		70:	
			N70 := REAL_TO_WORD (rLitros);
		80:	
			N80 := REAL_TO_WORD (rLitros);	
		90:	
			N90 := REAL_TO_WORD (rLitros);
		100:	
			N100 := REAL_TO_WORD (rLitros);	
	END_CASE
END_IF

/// Activar salida de llenado
xLlenado:= xInicioCalibracion AND (wNivel<100) AND NOT xPause ;

// Fin Calibracion
TP_FinCalibracion(IN:= xStart AND xInicioCalibracion AND (wNivel>=100) , PT:= T#1S, Q=> , ET=> );
xFinCalibracion:= TP_FinCalibracion.Q;

END_FUNCTION_BLOCK

// POUs/PLC/MC/Elements/fBCntLiters
FUNCTION_BLOCK fBCntLiters
VAR_INPUT
	xActv: BOOL;		/// Activate the counter
	xReset: BOOL;		/// Reset the liters value
	rInLiters: REAL;	/// Liters Input
END_VAR
VAR_OUTPUT
	rLiters: REAL;	/// Actual value 
END_VAR
VAR
	pResetLitros: R_TRIG;
	pInicio: R_TRIG;
	LitrosAcum: REAL;
END_VAR
VAR RETAIN
	/// Litros acumulados
	LitrosAc: REAL;
	/// Litros Inicial
	LitrosIni: REAL;
END_VAR

pInicio(CLK:=xActv );
//CARGAR LITROS INICIO
IF Pinicio.Q THEN
	LitrosIni := rInLiters;
	LitrosAcum:=rLiters;
END_IF

//CALCULAR LITROS EN PERIODO ACTIVO
IF xActv THEN
	LitrosAc := rInLiters-LitrosIni;
END_IF

//cALCULO LITROS
	rLiters := LitrosAc + LitrosAcum;


//PULSO RESET
pResetLitros(CLK:=xReset );
//rESET VALORES ACUMULADOS
IF  pResetLitros.Q THEN
	LitrosAcum := 0;	
	LitrosAc := 0;
	LitrosIni := 0;
END_IF

END_FUNCTION_BLOCK

// POUs/PLC/MC/Elements/fBHorn
FUNCTION_BLOCK fBHorn
VAR_INPUT
	axAlarm: ARRAY[1..Max_Alarmes] OF BOOL;
	axHorn: ARRAY[1..Max_Alarmes] OF BOOL;
	xStopHorn: BOOL;
END_VAR
VAR_OUTPUT
	xAlarmActv: BOOL;
	xHornActv: BOOL;
END_VAR
VAR
	iPunt: INT;
	afPulseAlarm: ARRAY[1..max_Alarmes] OF R_TRIG;
	xActvHorn: BOOL;
	fRS_Horn: Rs;
END_VAR


(*Comprobar si hay alarma activa*)
iPunt:=1;
xAlarmActv:=FALSE;
WHILE xAlarmActv=FALSE AND iPunt<WORD_TO_INT(Max_Alarmes)
	DO
	IF axAlarm[iPunt]=TRUE THEN
		xAlarmActv:=TRUE;
	END_IF
	iPunt:=iPunt+1;
END_WHILE


(*Activa o Reactiva Sirena*)

(*Pulso al Activar Sirena*)
iPunt:=1;
xActvHorn:=FALSE;
WHILE iPunt<WORD_TO_INT(Max_Alarmes) AND xActvHorn=FALSE
	DO
	afPulseAlarm[iPunt](CLK:= axHorn[iPunt]);
	xActvHorn:=afPulseAlarm[iPunt].Q AND xAlarmActv;
	iPunt:=iPunt+1;
END_WHILE
(*Marcha-Paro Sirena*)
fRS_Horn(SET:= xActvHorn, RESET1:=xStopHorn OR NOT(xAlarmActv));
xHornActv:=fRS_Horn.Q1;

END_FUNCTION_BLOCK

// POUs/PLC/MC/Elements/fbLiterCounter_by_flow
FUNCTION_BLOCK fbLiterCounter_by_flow
(*************************************************************
Convert a flow input into liters - 01/12/2021
V1.00
*************************************************************)
VAR_INPUT
	xActive : BOOL;			// Active the function
	rFlow :   REAL;			// Flow Input (l/min)
END_VAR
VAR_OUTPUT
	rLiters :   REAL;		// Liter output (REAL)
	dwLiters : 	DWORD;		//	Liter output (DDWORD)
END_VAR
VAR
	LitersSum : REAL;
	Periodecicle:Tcicle;
	ov: BOOL;
	INTEG: INTEGRAL;	
END_VAR


INTEG(
	IN:=rFlow , 
	TM:=10 , 
	RESET:=ov OR NOT xActive , 
	OUT=> LitersSum, 
	OVERFLOW=>ov );
	
rLiters := LitersSum/60;
dwLiters := REAL_TO_DWORD(LitersSum/60);

END_FUNCTION_BLOCK

// POUs/PLC/Utils/FreqCycle/TCicle
FUNCTION_BLOCK Tcicle
(**********************************************************
 - 29/11/2021
V1.00
*********************************************************)
VAR_INPUT

END_VAR
VAR_OUTPUT
	dwPeriode_Cicle:DWORD;		// Cycle Peryod
END_VAR

VAR_IN_OUT

END_VAR

VAR
	tempo: TON;
	reset: BOOL;
	t_actual: TIME;
	t_anterior: TIME;
	Periode: TIME;
END_VAR

tempo(IN:=NOT reset , PT:=T#7D , Q=>reset , ET=>t_actual );

Periode:= T_actual-T_anterior;

IF	NOT reset
	THEN
		T_anterior := T_actual;
END_IF

dwPeriode_cicle := TIME_TO_DWORD(Periode);

END_FUNCTION_BLOCK

// POUs/PLC/MC/Elements/fbLitersbyLevel
FUNCTION_BLOCK fbLitersbyLevel
(**********************************************
Convert an Level input into Liters - 01/12/2021
V1.00
***********************************************)
VAR_INPUT
	rLevel:REAL;
	dwN0:DWORD;
	dwN10:DWORD;
	dwN20:DWORD;
	dwN30:DWORD;
	dwN40:DWORD;
	dwN50:DWORD;
	dwN60:DWORD;
	dwN70:DWORD;
	dwN80:DWORD;
	dwN90:DWORD;
	dwN100:DWORD;
END_VAR
VAR_OUTPUT
	rLiters:REAL;
END_VAR
VAR
	iLiters:INT;
	LitrosMaq: CHARCURVE;
	litrosNivell:ARRAY[0..10]OF point;
END_VAR


litrosNivell[0].X := 0;
litrosNivell[0].Y := DWORD_TO_INT(dwN0);
litrosNivell[1].X := 100;
litrosNivell[1].Y := DWORD_TO_INT(dwN10);
litrosNivell[2].X := 200;
litrosNivell[2].Y := DWORD_TO_INT(dwN20);
litrosNivell[3].X := 300; 
litrosNivell[3].Y := DWORD_TO_INT(dwN30);
litrosNivell[4].X := 400;
litrosNivell[4].Y := DWORD_TO_INT(dwN40);
litrosNivell[5].X := 500;
litrosNivell[5].Y := DWORD_TO_INT(dwN50);
litrosNivell[6].X := 600;
litrosNivell[6].Y := DWORD_TO_INT(dwN60);
litrosNivell[7].X := 700;
litrosNivell[7].Y := DWORD_TO_INT(dwN70);
litrosNivell[8].X := 800;
litrosNivell[8].Y := DWORD_TO_INT(dwN80);
litrosNivell[9].X := 900;
litrosNivell[9].Y := DWORD_TO_INT(dwN90);
litrosNivell[10].X := 1000;
litrosNivell[10].Y := DWORD_TO_INT(dwN100);

LitrosMaq(
	IN:= REAL_TO_INT(rLevel*10) , 
	N:= 11, 
	P:= litrosNivell, 
	OUT=> iLiters, 
	ERR=> );

rLiters := INT_TO_REAL (iLiters);

END_FUNCTION_BLOCK

// POUs/PLC/MC/Elements/fbMeterCounter_by_Speed
FUNCTION_BLOCK fbMeterCounter_by_Speed
(*************************************************************
Convert an speed input into meters - 01/12/2021
V1.00
*************************************************************)
VAR_INPUT
	xMachineRunning:BOOL;
	xFabricPresence:BOOL;
	xReset:BOOL;
	rSpeed:REAL;
END_VAR
VAR_OUTPUT
	rMeters:REAL;
END_VAR
VAR
	ContarMetros: BOOL;
	Acumulador: ContadorRapid;
	cumulado: BOOL;
	acumulado: REAL;
	acumuladoInicial: REAL;
	acumuladofinal: REAL;
	Pulsocontador: F_TRIG;
	Acumular: BOOL;
END_VAR

ContarMetros := xMachineRunning AND xFabricPresence;

Pulsocontador(CLK:=ContarMetros , Q=>Acumular);

IF Acumular
	THEN
		acumuladoInicial := acumuladofinal;
END_IF

IF xReset
	THEN
		acumuladoInicial :=0;
		acumuladofinal :=0;
END_IF

Acumulador(bActivate:=ContarMetros AND NOT xReset , rFequency:=rSpeed , rCounter_REAL=>acumulado , dwCounter_DWORD=> );

acumuladofinal := acumulado + acumuladoInicial;

rMeters := acumuladofinal/60;

END_FUNCTION_BLOCK

// POUs/PLC/Utils/Counters/ContadorRapid
FUNCTION_BLOCK ContadorRapid
(**********************************************************
Creat an totalizer from an frequency input - 26/11/2021
V1.00
*********************************************************)
VAR_INPUT
	bActivate:BOOL;			// Start executing the function
	rFequency:REAL;			// Input Frequency
END_VAR

VAR_OUTPUT
	rCounter_REAL:REAL;
	dwCounter_DWORD:DWORD;
END_VAR

VAR
	Periodecicle:Tcicle;
	ov: BOOL;
	INTEG: INTEGRAL;
END_VAR



INTEG(
	IN:=rFequency , 
	TM:=Periodecicle.dwPeriode_Cicle , 
	RESET:= ov OR NOT bActivate , 
	OUT=> rCounter_REAL, 
	OVERFLOW=> ov);

dwCounter_DWORD := REAL_TO_DWORD(rCounter_REAL);

END_FUNCTION_BLOCK

// POUs/PLC/MC/Elements/fbPulseTrain
FUNCTION_BLOCK fbPulseTrain
(******************************************************
Generate a Pulse Train based on a % input - 12/01/2024
V1.02
*******************************************************)
VAR_INPUT
	rPorcentatge: REAL;		/// Percentual Input (0-100%)
	rPeriode_seg: REAL;		/// Period Input (sec)
	rPols_min_ms: REAL;		/// Minimum duration of the pulse output (ms)
END_VAR
VAR_OUTPUT
	xT_Pulsos: BOOL;		/// Pulse Output
END_VAR
VAR
	PararTren: BOOL;
	SegonsOFFtime: TIME;
	SegonsONtime: TIME;
	SegonsONreal: REAL;
	SegonsOFFreal: REAL;
	AperturaPulso: REAL;
	SegonsCicles: REAL;
	Tiemposinsenal: TMP;
	tempsmin: TIME;
	toff: TON;
	TON: TON;
	PulsMin: BOOL;
	TPulsMin: TP;
END_VAR

AperturaPulso := rPorcentatge;
SegonsCicles := rPeriode_seg;

SegonsONreal := (SegonsCicles*AperturaPulso)/100;

//no fer pols mes petit de pols minim en ON
IF SegonsONreal< (rPols_min_ms/1000)
	THEN
	SegonsONreal:=0;
END_IF
//no fer pols mes petit de pols minim en ON
IF SegonsONreal> SegonsCicles-(rPols_min_ms/1000)
	THEN
	SegonsONreal:=SegonsCicles;
END_IF

//CAlcular  temps OFF
SegonsOFFreal := SegonsCicles-SegonsONreal;

SegonsONtime := REAL_TO_TIME(SegonsONreal*1000);
SegonsOFFtime := REAL_TO_TIME(SegonsOFFreal*1000);


// Generador de pulsos
toff(IN:= NOT ton.Q, PT:=SegonsOFFtime , Q=> , ET=> );
ton(IN:= toff.Q, PT:=SegonsONtime , Q=> , ET=> );


xT_Pulsos := (toff.Q AND NOT PararTren) ;

END_FUNCTION_BLOCK

// POUs/PLC/MC/Elements/fBUp_Down
FUNCTION_BLOCK fBUp_Down
VAR_INPUT
	///Pulsador Subir 
	xUP: BOOL;
	///Pulsador Bajar 
	xDOWN: BOOL;
	///Velocidad para subir o bajar velocidad =100
	iFactor: INT := 100;
	rLimInf: REAL := 0;
	rLimSup: REAL := 100;
END_VAR
VAR_IN_OUT
	///Variable 
	SP: REAL;
END_VAR
VAR
	b_BaseTime: Blink;
	p_BaseTime: R_trig;
	xPulPulsado: BOOL;
	t2seg: Ton;
	t5seg: Ton;
	rFact: REAL;
	temps1: TIME := TIME#2s0ms;
	temps2: TIME := TIME#5s0ms;
	rFact1: REAL := 2.0;
	rFact2: REAL := 4;
END_VAR


(*Generar Base de tiempo par las subidad o bajadas*)
b_BaseTime(ENABLE:=TRUE , TIMELOW:=T#100MS , TIMEHIGH:=T#100MS , OUT=> );
p_BaseTime(CLK:=b_BaseTime.OUT );

(*Calcular Constante de subir o bajar *)
xPulPulsado:= xUP OR xDown;
t2seg(IN:=xPulPulsado , PT:=temps1  );
t5seg(IN:=xPulPulsado , PT:=temps2  );

IF NOT(t2seg.Q)
	THEN
	rFact:=INT_TO_REAL(iFactor)/100.0;
	ELSIF t2seg.Q AND NOT(t5seg.Q)
		THEN
		rFact:=INT_TO_REAL(iFactor)*rFact1/100.0;
		ELSIF t5seg.Q
			THEN
				rFact:=INT_TO_REAL(iFactor)*rFact2/100.0;
END_IF


(*Subir consigna*)
IF xUP AND p_BaseTime.Q
	THEN
	SP:=SP+rFact;
END_IF

(*Bajar consigna*)
IF xDOWN AND p_BaseTime.Q
	THEN
	SP:=SP-rFact;
END_IF

(*Limite Superior*)
IF SP>rLimSup THEN
	SP:=rLimSup;
END_IF

(*Limite Inferior*)
IF SP<rLimInf THEN
	SP:=rLimInf;
END_IF

END_FUNCTION_BLOCK

// POUs/PLC/MC/Elements/fbWashing_HT
FUNCTION_BLOCK fbWashing_HT
(**************************************************************
Execute a continuos washing in high temperature - 01/12/2021
V1.00
***************************************************************)
VAR_INPUT
	xStartDrain : BOOL;					// Enable the function
	xDirectDrain:BOOL;					// Enable direct drain input
	dwTimeFillAuxTank: DWORD;			// Time to transfer from machine to auxiliar tank
	dwTimeCloseAuxTank:DWORD;			// Time to finish the transfering to the auxiliar tank
	dwTimeDepAuxTank:DWORD;				// Time do depressurize auxiliar tank
	dwTimeDrainAunxTank:DWORD;			// Time to drain the auxiliar tank
	dwTimeCloseDrainAuxTank:DWORD;		// Time to garantee that the drain valve has closed
	xAlarmPauseWash:BOOL;				// Alarm Input to stop the function
	
END_VAR

VAR_OUTPUT
	xFillAuxTank:BOOL;					// Transfer from machuine to auxiliar tank
	xDepAuxTank:BOOL;					// depressurize auxiliar tank
	xDrainAuxTank:BOOL;					// Drain auxiliar tank
END_VAR

VAR
	ObrirBuidatRBB: BOOL;
	TempoPas1: TMP;
	TempoPas2: TMP;
	ObrirDespresuritzaRBB: BOOL;
	TempoPas3: TMP;
	ObrirOmplertaRBB: BOOL;
	TancarOmpertaRBB: BOOL;
	TancarBuidatRBB: BOOL;
	FiSequenciaRBB: BOOL;
	TempoPas4: TMP;
	TempoPas5: TMP;
	TemoDespesuritzaRBB: TMP;
	RBBsensePresio: BOOL;
	ObrirRespiraderoRBB: BOOL;
	FiBuidatRBB: BOOL;
	FiBuidatDirecte: F_TRIG;
	PolsFiBuidat: BOOL;
	TempSfINAL: TMP;
	ObrirBuidatAlBuidat: BOOL;
	srObrirOmplertaRBB :SR;
	srObrirRespiraderoRBB:SR;
	srPolsFiBuidat:SR;
	rtBuidatDirecte:F_TRIG;
	
	
END_VAR

// **************** Inicia el ciclo **************************
srObrirOmplertaRBB(SET1:= xStartDrain AND NOT srObrirOmplertaRBB.Q1 , RESET:=xAlarmPauseWash OR (FiSequenciaRBB AND ObrirOmplertaRBB) , Q1=>ObrirOmplertaRBB );


// **************** Temps por cada pas ************************
TempoPas1(xIN:=ObrirOmplertaRBB , dwSegons:=dwTimeFillAuxTank , xQ=>TancarOmpertaRBB , dwTsegons=> );

TempoPas2(xIN:=TancarOmpertaRBB , dwSegons:=dwTimeCloseAuxTank , xQ=>ObrirDespresuritzaRBB , dwTsegons=> );

TempoPas3(xIN:=ObrirDespresuritzaRBB , dwSegons:=dwTimeDepAuxTank , xQ=>ObrirBuidatRBB , dwTsegons=> );

TempoPas4(xIN:=ObrirBuidatRBB , dwSegons:=dwTimeDrainAunxTank , xQ=>TancarBuidatRBB , dwTsegons=> );

TempoPas5(xIN:=TancarBuidatRBB , dwSegons:=dwTimeCloseDrainAuxTank , xQ=>FiSequenciaRBB , dwTsegons=> );


srObrirRespiraderoRBB(SET1:=xDirectDrain AND NOT srObrirRespiraderoRBB.Q1, RESET:=xAlarmPauseWash OR (FiBuidatRBB AND ObrirRespiraderoRBB) , Q1=>ObrirRespiraderoRBB );

TemoDespesuritzaRBB(xIN:=ObrirRespiraderoRBB , dwSegons:=dwTimeDepAuxTank , xQ=>RBBsensePresio , dwTsegons=> );

rtBuidatDirecte(CLK:=xDirectDrain , Q=> );
srPolsFiBuidat(SET1:=rtBuidatDirecte.Q , RESET:=FiBuidatRBB , Q1=>PolsFiBuidat );

TempSfINAL(xIN:=PolsFiBuidat , dwSegons:=5 , xQ=>FiBuidatRBB , dwTsegons=> );

ObrirBuidatAlBuidat := xDirectDrain AND NOT FiBuidatRBB;

///*************************** Activa salidas ******************************
xFillAuxTank := (ObrirOmplertaRBB AND NOT TancarOmpertaRBB AND NOT xAlarmPauseWash) OR (xDirectDrain AND RBBsensePresio);

xDepAuxTank := (ObrirDespresuritzaRBB AND NOT TancarBuidatRBB AND NOT xAlarmPauseWash) OR xDirectDrain;

xDrainAuxTank := (ObrirBuidatRBB AND NOT TancarBuidatRBB AND NOT xAlarmPauseWash) OR ObrirBuidatAlBuidat;

END_FUNCTION_BLOCK

// POUs/PLC/MC/Fill/fBTemperatureFill
FUNCTION_BLOCK fBTemperatureFill
VAR_INPUT
	///Enable the temperature control
	xActiv: BOOL;
	/// Temperature SetPoint
	rTempSP: REAL;
	/// Real Temperature 
	rTempPV: REAL;
	/// Superior DeadBand 
	rDBHigh: REAL;
	/// Inferior DeadBand 
	rDBLow: REAL;
	///	Maximum time for adjust the temperature
	timMaxTime: TIME;
	///	Maximum time configure (1 - Open just cold water, 0 - Open cold and hot water, 2 - Activate Alarm)
	dwConfigMaxTime: DWORD;
	/// Minimum level input
	xLevel: BOOL;
	/// Level Configure (0 - Disable, 1 - Starts filing with CW and HW, 2 - Starts filing with CW, 3 - Starts filing with HW) 
	dwConfigLevel: DWORD;
	/// Time delay for start adjusting the teperature.
	timControl: TIME;
END_VAR
VAR_OUTPUT
	/// Cold Water Output
	xCWater: BOOL;
	/// Hot Water Output
	xHWater: BOOL;
	/// Maximum time alarm Output
	xAlarmMaxTime: BOOL;
END_VAR
VAR
	TempIni: TON;
	MaxTemp: TON;
	/// Temperatura mínima SP-DBmin	
	TemperMin: REAL;
	/// Temperatura mínima SP+DBmax
	TemperMax: REAL;
	CtrlNivel: BOOL;
	xNivOK: BOOL;
	xRegOutDB: BOOL;
END_VAR


//Delay para empezar la regulacion
TempIni(IN:=xActiv, PT:=timControl , Q=> , ET=> );

//Esperar nivel minimo si es necesario
IF dwConfigLevel > 0
	THEN
		xNivOK := xLevel;
	ELSE
		xNivOK := 1;
END_IF

//Margenes de la banda muerta de regulacion			
TemperMax := rTempSP + rDBHigh;
TemperMin := rTempSP - rDBLow;
//Temperatura Fuera banda muerta
xRegOutDB:=  ((rTempPV < TemperMin) OR (rTempPV > TemperMax));

//Tiempo maximo de regulacion
MaxTemp(	IN:=	TempIni.Q AND 						//inicia reguñacion
					xRegOutDB AND 						//Temperatura fuera banda muerta
					xNivOK  , 							//Esperar si es necesario el nivel 
			PT:=	timMaxTime ,						//tiempo maximo de regulacion 
			Q=>		xAlarmMaxTime );					//Alarma tiempo maxioms reg

			

IF xActiv
	THEN
		//Abrir 2 aguas
		IF (xRegOutDB AND (NOT MaxTemp.Q)) OR      //temp fuera banda muerta
			(MaxTemp.Q AND (dwConfigMaxTime = 0) AND (dwConfigMaxTime <> 2)) OR 
			NOT(TempIni.Q) OR 
			(dwConfigLevel = 1 AND NOT xLevel) 
			THEN
				xCWater :=TRUE;
				xHWater :=TRUE;
		END_IF	
		IF 	rTempPV > TemperMax AND 
			NOT(MaxTemp.Q) AND 
			(	TempIni.Q OR 
				(MaxTemp.Q AND dwConfigMaxTime = 1 AND dwConfigMaxTime <> 2) OR 
				(dwConfigLevel = 3 AND NOT xLevel)
			)
			THEN			
				xCWater :=TRUE;
				xHWater :=FALSE;			
		END_IF 
		IF rTempPV < TemperMin AND 
		NOT(MaxTemp.Q) AND 
		(	TempIni.Q OR 
			(dwConfigLevel = 2 AND NOT xLevel)
		)
			THEN			
				xCWater :=FALSE;
				xHWater :=TRUE;			
		END_IF
		IF MaxTemp.Q AND dwConfigMaxTime = 2
			THEN
				xCWater :=FALSE;
				xHWater :=FALSE;
		END_IF
	 ELSE
		xCWater :=FALSE;
		xHWater :=FALSE;			
END_IF

END_FUNCTION_BLOCK

// POUs/PLC/MC/Pump/fBPumpC
FUNCTION_BLOCK fBPumpC
VAR_INPUT
	///Pulsador de marcha
	fP_Run: BOOL;
	///Pulsador de paro
	fP_Stop: BOOL;
	///Pulsador de continua programa
	xP_ContProg: BOOL;
	///Nivel Seguridad Bomba
	xLvlSeg: BOOL;
	///Condiciones Seguridad arranque Bomba
	xSeg: BOOL;
	///Condiciones arrancar Bomba
	xConditionRun: BOOL;
	/// Condiciones paran bomba
	xConditionStop: BOOL;
	///1:manual  2: auto
	iAutoMan: INT;
END_VAR
VAR_OUTPUT
	Run: BOOL;
END_VAR
VAR
	xExistePulParo: BOOL;
	RT_PasoAuto: R_trig;
	xRunForPul: BOOL;
	RT_Run: R_trig;
	RT_Stop: R_trig;
	xStopForPul: BOOL;
	xArrancar: BOOL;
	xRunContProg: BOOL;
	tContProg: Ton;
	xParar: BOOL;
	RS_PUMP: Rs;
	a: INT;
	FTParoPorNoMarcha: F_TRIG;
	xParoPorNoMarcha: BOOL;
	TON_MarchaBomba: TON;
END_VAR

a:=a+1;

(*-------------------------------------------*)
(****** Condiciones de Inicio******)
//Con pulsación de 1 segundo funciona como pulsador de marcha
//Con pulsación de más de 1 segundo funciona como barra (selector)*) 

(*-----Gestion Pulsadores-----*)

(*Pulso Run*)
RT_Run(CLK:=fP_run );

(*Pulso Stop*)
RT_Stop(CLK:=fP_Stop );

(*Pulso Paro por no marcha*)
TON_MarchaBomba(IN:= fP_run, PT:= T#1S, Q=> , ET=> );
FTParoPorNoMarcha(CLK:=TON_MarchaBomba.Q , );

xParoPorNoMarcha:= FTParoPorNoMarcha.Q;

(*Pul Cont Prog,*)
tContProg(IN:=xP_ContProg , PT:=T#5S);


(*-----Paso a Auto------*)
RT_PasoAuto(CLK:= iAutoMan=2 );


(*------------------------------------*)
(*     Marcha       *) 
(*------------------------------------*)
xArrancar:= RT_Run.Q OR  			(*Arranc pulsadors*)
			tContProg.Q OR  		(*Arranc Cont Prog*)	
			RT_PasoAuto.Q OR
			xConditionRun;
			
			
(*------------------------------------*)
(*     Paro       *) 
(*------------------------------------*)
xParar:= 	RT_Stop.Q OR 			(*Paro  por pulsadores*)
			xConditionStop OR		(*Condiciones de paro*)
			//NOT(xLvlSeg) OR			(*Falta nivel de seguridad*)
			NOT(xSeg)OR
			xParoPorNoMarcha;    (*Paro cuando salimos de marcha con barra*)
			
(*------------------------------------*)
(*     Arranque       *) 
(*------------------------------------*)
			
RS_PUMP(SET:=xArrancar , RESET1:= xParar );

Run:= 	RS_pump.Q1;

END_FUNCTION_BLOCK

// POUs/PLC/MC/Pump/fBPumpSpeed
FUNCTION_BLOCK fBPumpSpeed
VAR_INPUT
	///Bomba en marcha
	xRun: BOOL;
	///0=Man  1=Auto  
	xAutoMan: BOOL;
	///Pulsador Subir Velocidad
	xUP_Speed: BOOL;
	///Pulsador Bajar Velocidad
	xDOWN_Speed: BOOL;
	///Consigna de la funcion velocidad 0..100%
	rSP_Function: REAL;
	iFACTOR: INT := 50;
END_VAR
VAR_OUTPUT
	///Consigna velocidad 0..100%
	SP_Speed: REAL;
	///Consigna velocidad Auto 0..100%
	SP_Auto: REAL;
	///Consigna velocidad Manual 0..100%
	SP_Man: REAL;
END_VAR
VAR
	GestPul: fBUP_down;
	a: INT;
END_VAR

a:=a+1;
(*GESTION SP MANUAL*)
(*cargar valor sp auto al estar en auto*)
IF (xAutoMan) THEN
	SP_Man:=SP_Auto;
END_IF

(*GESTION SP AUTO*)
SP_Auto:=rSP_Function;


(*Gestion Pulsadores*)
GestPul(
	xUP:= 		xUP_Speed, 
	xDOWN:= 	xDOWN_Speed, 
	iFactor:= 	iFACTOR, 
	rLimInf:= 	0, 
	rLimSup:= 	100, 
	SP:= SP_Man);

(*Gestion SP*)

IF xAutoMan 
	THEN
	SP_Speed:=SP_Auto;
	ELSE
	SP_Speed:=SP_Man;		
END_IF

IF NOT(xRun) 
	THEN
	SP_Speed:=0;
END_IF

END_FUNCTION_BLOCK

// POUs/PLC/MC/Seam/fBSeamTime
FUNCTION_BLOCK fBSeamTime
VAR_INPUT
	xWinchRun: BOOL;
	xControlActv: BOOL;
	xSeamDetect: BOOL;
	iPercContol: INT;
	iTimeMax: INT;
END_VAR
VAR_OUTPUT
	xStoped: BOOL;
	xCntrlRun: BOOL;
	xNoSeam: BOOL;
	xDetectionPulse: BOOL;
	iTimeAct: INT;
	iTimeAnt1: INT;
	iTimeAnt2: INT;
	iTimeAnt3: INT;
END_VAR
VAR
	///Durada del 
	tTimePulseOut: TIME := TIME#2s0ms;
	tTimePulseMin: TIME := TIME#200ms;
	tTimerMinPulse: ton;
	pPulseSeam: r_trig;
	TTimerPulse: tp;
	tTimerSeam: ton;
	iPasesParacontrol: INT := 2;
	cContPaso: CTU;
	tTimeAlarm: REAL;
	xBloqPulso: BOOL;
	tTimeMax: TIME;
END_VAR



//Asegurar un pulso minimo par descartar rebotes
tTimerMinPulse(IN:=xSeamDetect , PT:=tTimePulseMin );
pPulseSeam(CLK:=tTimerMinPulse.Q);

//Generar Pulso de deteccion con tiempo fijo
TTimerPulse(IN:= pPulseSeam.Q, PT:=tTimePulseOut );
xDetectionPulse:= TTimerPulse.Q  ;

//Bloquear pulsos por posible rebote
xBloqPulso:= (iTimeAct<(iTimeAnt1/20));

//Acumular temps de pas al detectar pas d'iman
IF xWinchRun AND pPulseSeam.Q AND NOT(xBloqPulso)
	THEN
		iTimeAnt3:=iTimeAnt2;
		iTimeAnt2:=iTimeAnt1;
		iTimeAnt1:=iTimeAct;
END_IF

//Calculo tiempo actual
tTimerSeam(	IN:=xWinchRun AND NOT(pPulseSeam.Q) AND xControlActv, 
			PT:=T#1D );

iTimeAct:=TIME_TO_INT(tTimerSeam.ET/1000);



//Control Paso de cuerda

cContPaso(
	CU:= 		xControlActv AND pPulseSeam.Q , 
	RESET:= 	NOT(xControlActv), 
	PV:= 		INT_TO_WORD(iPasesParacontrol));
	
xCntrlRun:=cContPaso.Q;

//Tiempo maximo calculado con el porcentaje
tTimeAlarm:= (INT_TO_REAL(iTimeAnt1)*(1.0+INT_TO_REAL(iPercContol)/100.0))  ;


xStoped:= 	xCntrlRun AND				//control activo
			cContPaso.Q AND 			//La cuerda ha pasado 2 veces
			(iTimeAct >	tTimeAlarm);	//tiempo actual mayor al anterior	
			
//Alarma de FALTA IMAN (xNoSeam)			
xNoSeam:= 	xCntrlRun AND				//control activo
			xWinchRun AND 				//Torniquete en marcha
			(iTimeAct >	iTimeMax);		//tiempo actual mayor el Maximo

END_FUNCTION_BLOCK

// POUs/PLC/MC/Temperature/fBTermo
FUNCTION_BLOCK fBTermo
VAR_INPUT
	///		Activa el calcul del gradient
	TermoActv: BOOL;
	///		Lectura de la temperatura 
	TemperaturaReal: REAL;
	///		Temperatura final que es vol obtenir  
	TemperaturaFinal: REAL;
	///		Expresat en decimes de grau 
	Gradient: REAL;
	///		Temps de maneniment en minuts 
	t_Manteniment: REAL;
	///		Entrada que s'utilitza com a rellotge (1seg per regular per temps) 
	Pols: BOOL;
	///		Aquesta entrada produeix una pausa en el calcul 
	PausaExterior: BOOL;
	///		Diferencia de temperatura necesaria per parar la consigna per 
	///		esperar a la temperatura real. Definit en  graus, per defecte =2  
	GrausPerIntegracio: REAL := 2;
	///		Diferencia de graus amb les que es forzara calentar encara que la
	///		temperatura sigui superior i la consigna pasarà a ser directament 
	///		la temperatura final .definit en graus i real. per defecte =4  
	GrausForzarCal: REAL := 4;
	///		Recomença la termoregulacio agafant la temperaturaimposada 
	///		com a inicial.  S'utilitza per poder modificar el gradient en una 
	///		introducció ( fa un reset a la durada i agafa el gradient actual). 
	ReIniciarTermo: BOOL;
	///		Temps seguretat per a cambiar de calentar a refredar o al reves
	///		 per defecte =30
	TmoSegConmutacion: DWORD := 30;
	///		diferencia de teperatura per realitzar la conmutació durant 
	///		el manteniment  per defecte =5
	ConmutacioEnManteniment: REAL := 5;
	BandaProporcional: REAL;
	PartIntergral: REAL;
	PartDerivada: REAL;
	T_periode: REAL;
	SeguretatOK: BOOL;
	ObrirPurgaenRepos: BOOL;
	t_Purga: DWORD;
	///Paralel: Temperatura per iniciar el calcul de la termorregulacio 
	TemperaturaPerInici: REAL;
	NO_Reset: BOOL;
END_VAR
VAR_OUTPUT
	///		Indica que la termorregulacio esta pausada per integracio
	EnIntegracio: BOOL;
	///		Indicacio de la temperatura imposada
	TemperaturaImposada: REAL;
	///		Termoregulació per calentar, Es la ordre al regulador
	Vapor: BOOL;
	Apertura_Vapor: REAL;
	///		Termoregulació per refredar, , Es la ordre al regulador 
	AiguaRefredament: BOOL;
	Apertura_Refreda: REAL;
	///		Indicacio que la temperatura a arribat a la temperatura final 
	EnManteniment: BOOL;
	Actv_RetornAigua: BOOL;
	Actv_RetornVapor: BOOL;
	Actv_BuidatSerpenti: BOOL;
	DuradaTermo: DWORD;
	///solo informacion
	refredar: BOOL;
	///solo informacion
	calentar: BOOL;
END_VAR
VAR
	TemperaturaInicial: REAL;
	TemporIniciar: TON;
	IniciarTermo: BOOL;
	TempsEnMarxa: BOOL;
	DiferencialImposada: REAL;
	DiferenciaTemp: REAL;
	ActvManteniment: BOOL;
	TempoManteniment: TON;
	errorPID: BOOL;
	ResetPID: BOOL;
	EsperaSortida: BOOL;
	OKCalentar: TMPPausa;
	OKRefredar: TMPPausa;
	TemperaturaMaxima: REAL;
	TemperaturaMinima: REAL;
	TempsTempAlta: TON;
	PasarARefredar: BOOL;
	TempsTempBaixa: TON;
	PasarACalentar: BOOL;
	Part_Proporcional: REAL;
	PI: REAL;
	Y_min: REAL;
	Y_max: REAL;
	PID_CALENTAR: PID_fixcycle;
	polsResetMant: R_TRIG;
	ResetGrad0: BOOL;
	SortidaPID: REAL;
	tempsPurga: TMPPausa;
	TR: REAL;
	TI: REAL;
	Actv_Vapor: BOOL;
	Actv_AiguaRefredament: BOOL;
	PI_reg: REAL;
	xMan: BOOL := FALSE;
	xLim: BOOL;
	xOver: BOOL;
	IN: INT;
	DE: TMPPausa;
	D: TON;
END_VAR

(*iniciar TermoRegulación*)
TemporIniciar
	(IN:= TermoActv ,
	 PT:= T#1s ,
	 Q=> IniciarTermo ,
	 ET=> );

(*Guardar valor temperatura inicial*)
IF NOT(IniciarTermo)
	THEN
		IF TemperaturaPerInici=0
			THEN
			TemperaturaInicial:=TemperaturaReal;
			DuradaTermo:=0;
			ELSE
			TemperaturaInicial:=TemperaturaPerInici;
			DuradaTermo:=0;
		END_IF
END_IF


(*Reiniciar el calcul de la consigna de la termorregulacio*)
IF ReIniciarTermo
	THEN
		TemperaturaInicial:=TemperaturaImposada;
		DuradaTermo:=0;
END_IF


(*Termoregulacio  en integració*)
IF Calentar
	THEN
		DiferenciaTemp:=TemperaturaImposada - TemperaturaReal;
END_IF
IF Refredar
	THEN
		DiferenciaTemp:=TemperaturaReal-TemperaturaImposada;
END_IF
IF (DiferenciaTemp>GrausPerIntegracio) AND TermoActv
	THEN
		EnIntegracio:=TRUE;
	ELSE
		EnIntegracio:=FALSE;
END_IF

(*Calcul del  Temps de termoregulacio*)
TempsEnMarxa:= (IniciarTermo) AND NOT(PausaExterior) AND NOT(EnManteniment) AND NOT(EnIntegracio);
IF (TempsEnMarxa) AND (Pols)
	THEN
		DuradaTermo:=DuradaTermo+1;
END_IF

(* Mirar si calenta o refreda *)
IF TermoActv
	THEN
		IF ((TemperaturaFinal+GrausForzarCal) >= (TemperaturaInicial))
			THEN
				Calentar:= TRUE;
				Refredar:= FALSE;
		END_IF
		IF ((TemperaturaFinal+GrausForzarCal) < (TemperaturaInicial))
			THEN
				Calentar:= FALSE;
				Refredar:= TRUE;
		END_IF
	ELSE
		Calentar:= FALSE;
		Refredar:= FALSE;
END_IF

(*Calcul Tamperatura*)
IF Gradient<>0
	THEN
		DiferencialImposada:= ((Gradient * DWORD_TO_REAL(DuradaTermo)) / 600.0) ;
		IF calentar
			THEN
				TemperaturaImposada:= TemperaturaInicial+DiferencialImposada;
				IF TemperaturaImposada > TemperaturaFinal
				THEN
					TemperaturaImposada := TemperaturaFinal;
				END_IF
			ELSE
				IF refredar
					THEN
						TemperaturaImposada:= TemperaturaInicial - DiferencialImposada;
					ELSE
						TemperaturaImposada := TemperaturaReal;
				END_IF
		END_IF
	ELSE
		TemperaturaImposada := TemperaturaFinal;
END_IF
IF NOT(TermoActv)
	THEN
		TemperaturaImposada := TemperaturaReal;
END_IF


(*Calcular Si esta en manteniment*)
IF gradient<>0
	THEN
		IF ((TemperaturaImposada >= TemperaturaFinal AND Calentar) OR 
			(TemperaturaImposada <= TemperaturaFinal AND Refredar))
			THEN
				ActvManteniment:=TRUE;
				TemperaturaImposada:=TemperaturaFinal;
		END_IF
	ELSE
		IF ((TemperaturaReal >= (TemperaturaFinal-(GrausPerIntegracio) ) AND Calentar) OR (TemperaturaReal <= (TemperaturaFinal + (GrausPerIntegracio)) AND Refredar))
			THEN 
				ActvManteniment:=TRUE;
		END_IF
END_IF

IF NOT(TermoActv)
	THEN
		ActvManteniment:=FALSE;
END_IF

TempoManteniment(IN:= ActvManteniment, PT:= T#5S, Q=> , ET=> );

EnManteniment:=Tempomanteniment.Q;

(*@@@@@@@@@@@@@@@@@@@@@@@@@@@@@@@@@@@@@@@@@@@@@@@@@@@@@@@@@@@@@@@@@@@@*)


(*Si no calenta ni refreda es fa un reset del pid*)
(*Reset al entrar en manteniment*)
ResetGrad0:=((TemperaturaReal >= (TemperaturaFinal-(BandaProporcional/10.0) ) AND Calentar) OR (TemperaturaReal <= (TemperaturaFinal + (BandaProporcional/10.0)) AND Refredar));
polsResetMant(CLK:= ((gradient<>0 AND EnManteniment AND NOT(no_reset)) OR (gradient=0 AND ResetGrad0))); 			(*24/05/2013 modificat*)
IF (NOT(Calentar) AND NOT(Refredar)) OR (errorPID)  OR  (polsResetMant.Q) OR pasaraCalentar OR PasaraRefredar
	THEN
		ResetPID:=TRUE;
	ELSE
		ResetPID:=FALSE;
END_IF

(*Seguretat per activar el calentament*)

OKCalentar(
		xIN:= NOT(Refredar), 
		xPausa:= FALSE, 
		dwSegons:= TmoSegConmutacion , 
		xQ=> , 
		dwTsegons=> , 
		rTsegons=> );

OKRefredar(
		xIN:= NOT(Calentar), 
		xPausa:= FALSE, 
		dwSegons:= TmoSegConmutacion , 
		xQ=> , 
		dwTsegons=> , 
		rTsegons=> );

(*Activar Calentar o Refredar  tenint en compte el mantnment*)
(*Manteniment NO actiu*)
EsperaSortida:= (EnManteniment AND ((calentar AND okcalentar.xQ) OR (refredar AND okrefredar.xQ)));
IF NOT(EnManteniment) OR NOT EsperaSortida
	THEN
		Actv_Vapor :=Calentar AND okcalentar.xQ;
		Actv_AiguaRefredament :=Refredar AND okrefredar.xQ ;
END_IF
(*Manteniment SI actiu*)
(* Temperatures per fer les conmutacions *)
TemperaturaMaxima := TemperaturaImposada + (ConmutacioEnManteniment);
TemperaturaMinima := TemperaturaImposada - (ConmutacioEnManteniment);
(*Pasar  de calentar a refredar*)

TempsTempAlta(IN:= ((Actv_Vapor)AND(TemperaturaMaxima<TemperaturaReal)AND(EnManteniment)), 	
					PT:=T#5S , 
					Q=> PasarARefredar, ET=> );

IF PasarARefredar
	THEN
		Actv_Vapor:=FALSE;
		Actv_AiguaRefredament:=TRUE;
END_IF
(*Pasar  de refredar a calentar*)

TempsTempBaixa(IN:= ((Actv_AiguaRefredament)AND(TemperaturaMinima>TemperaturaReal)AND(EnManteniment)), 
					PT:= T#5S, 
					Q=> PasarACalentar, 
					ET=> );

IF PasarACalentar
	THEN
		Actv_Vapor:=TRUE;
		Actv_AiguaRefredament:=FALSE;
END_IF

(*Preparar valors del PID*)
(* BandaProporcional *)
IF BandaProporcional=0
	THEN
		BandaProporcional:=10.0;
END_IF
(*Calcul Part Proorcional*)
Part_Proporcional:=(1000.0/BandaProporcional);
(* Part integral*)
IF Gradient=0 AND NOT(enmanteniment)
THEN
PI:=0;
ELSE
PI:=PartIntergral;
END_IF
(*Maxim i minim *)
		Y_min:=0;
		Y_max:=100;
(*Temperatures PID*)
IF Actv_Vapor
	THEN
		TR:=TemperaturaReal;
		TI:=TemperaturaImposada;
END_IF
IF Actv_AiguaRefredament
	THEN
		TR:=300-TemperaturaReal;
		TI:=300-TemperaturaImposada;
END_IF

IF PI<=0 THEN
	PI_reg:=1E+36;
	ELSE
	PI_reg:=PI;	
	END_IF

PID_CALENTAR(
	ACTUAL:= 	TR, 
	SET_POINT:= TI, 
	KP:= 		Part_Proporcional, 
	TN:=		PI_reg , 
	TV:= 		PartDerivada, 
	Y_MANUAL:= 	0, 
	Y_OFFSET:= 	0, 
	Y_MIN:= 	Y_min, 
	Y_MAX:= 	Y_max, 
	MANUAL:= 	xMan, 
	RESET:= 	ResetPID, //Activar al cambiar el PID
	CYCLE:= 	0.01, 
	Y=> 		SortidaPID, 
	LIMITS_ACTIVE=> xLim, 
	OVERFLOW=> 		xOver);
	
	
	
(*	
PID_CALENTAR(
	ActValue:=TR ,
	SetPoint:= TI,
	Kp:= Part_Proporcional,
	Tn:= PI,
	Tv:=PartDerivada ,
	Ymin:=Y_min ,
	Ymax:=Y_max ,
	T:= T_periode,
	Normed:=1.0 ,
	Hold:=ResetPID ,
	Yman:=0 ,
	Yout=> SortidaPID);

*)
IF Actv_Vapor
	THEN
		Apertura_Refreda:=0;
		Apertura_Vapor:=SortidaPID;
END_IF
IF Actv_AiguaRefredament
	THEN
		Apertura_Refreda :=(SortidaPID);
		Apertura_Vapor:=0;
END_IF
(*Si no hi ha calentar o refredar parar-ho tot*)
(*Esposa al final per evitar que s'activin el les sortides per error*)
IF (Actv_Vapor=FALSE)AND(Actv_AiguaRefredament=FALSE)
	THEN
		Apertura_Vapor:=0.0;
		Apertura_Refreda:=0.0;
END_IF
(*================================================	*)
(*					SEGURETATS								*)
(*================================================	*)
IF NOT(SeguretatOK)
	THEN
		Vapor:=FALSE;
//		AiguaRefredament:=FALSE;
		Apertura_Vapor:=0.0;
//		Apertura_Refreda:=0.0;
ELSE
		Vapor:=Actv_Vapor;

END_IF
		AiguaRefredament:=Actv_AiguaRefredament;

(*================================================	*)
(*			retorno condensadors								*)
(*================================================	*)
(* Refredament *)
IF Actv_AiguaRefredament
	THEN
		Actv_RetornAigua:=TRUE;
		Actv_RetornVapor:=FALSE;
		Actv_BuidatSerpenti:=FALSE;
END_IF
(*calentament*)
tempsPurga(
		xIN:= Actv_Vapor, 
		xPausa:= FALSE, 
		dwSegons:= t_Purga, 
		xQ=> , 
		dwTsegons=> , 
		rTsegons=> );

IF Actv_Vapor AND NOT(tempsPurga.XQ)
THEN
		Actv_RetornAigua:=FALSE;
		Actv_RetornVapor:=FALSE;
		Actv_BuidatSerpenti:=TRUE;
END_IF
IF Actv_Vapor AND (tempsPurga.xQ)
THEN
		Actv_RetornAigua:=FALSE;
		Actv_RetornVapor:=TRUE;
		Actv_BuidatSerpenti:=FALSE;
END_IF
(*Repo*)
IF NOT(Actv_Vapor) AND NOT(Actv_AiguaRefredament) AND NOT(Actv_BuidatSerpenti)
THEN
		Actv_RetornAigua:=FALSE;
		Actv_RetornVapor:=FALSE;
		Actv_BuidatSerpenti:=FALSE;
END_IF
IF NOT(Actv_Vapor) AND NOT(Actv_AiguaRefredament) AND (Actv_BuidatSerpenti)
THEN
		Actv_RetornAigua:=FALSE;
		Actv_RetornVapor:=FALSE;
		Actv_BuidatSerpenti:=TRUE;
END_IF

END_FUNCTION_BLOCK

// POUs/PLC/Utils/AnalogConversions/Canvi_Escala
FUNCTION Canvi_Escala:REAL
(**************************************************************
Execute an SCALE from an input value (REAL). If not defined
 the scales, the default values are going to be 0 (min) and 100 (max)
for both, input and output. 26/11/2021
V1.00
***************************************************************)
VAR_INPUT
	rIn:REAL;						// Input Variable
	rIn_Min:REAL:=0;				// Input Low Value
	rIn_Max:REAL:=100;				// Input High Value
	rOut_Min:REAL:=0;				// Output Low Value
	rOut_Max:REAL:=100;				// Output High Value
END_VAR

VAR
	Din: REAL;
	Dout: REAL;
END_VAR

IF rin<rin_Min
	THEN
		rin:=rin_min;
END_IF
IF rin>rin_Max
	THEN
		rin:=rin_max;
END_IF

Din:=rIn_Max-rIn_Min;

IF Din=0
	THEN
		Canvi_Escala:=0;
	ELSE
		Dout:=rOut_Max-rOut_Min;
		Canvi_Escala:=(((rIn-rIn_Min)/Din)*Dout)+rOut_Min;
END_IF

END_FUNCTION

// POUs/PLC/Utils/AnalogConversions/Conv_Temp
FUNCTION Conv_Temp:REAL
(**************************************************************** 
 Convert an temperature input (INT * 10) to an REAL value (with decimals).  26/11/2021
 V1.00
*****************************************************************)
VAR_INPUT
	wLecturaTemperatura:WORD;				//Temperature Input (WORD)
END_VAR

VAR

END_VAR

Conv_Temp:= (WORD_TO_REAL(wLecturaTemperatura))/10;

END_FUNCTION

// POUs/PLC/Utils/BitsConversions/Bits_to_Dword
FUNCTION_BLOCK Bits_to_Dword
(**********************************************************
Join 32 bits in a DWORD Variable  - 29/11/2021
V1.0
*********************************************************)
VAR_INPUT
	bBB0:BOOL;		//LSB BYTE 0
	bBB1:BOOL;
	bBB2:BOOL;
	bBB3:BOOL;
	bBB4:BOOL;
	bBB5:BOOL;
	bBB6:BOOL;
	bBB7:BOOL;		//MSB BYTE 0
	bBA0:BOOL;		//LSB BYTE 1
	bBA1:BOOL;
	bBA2:BOOL;
	bBA3:BOOL;
	bBA4:BOOL;
	bBA5:BOOL;
	bBA6:BOOL;
	bBA7:BOOL;		//MSB BYTE 1
	bAB0:BOOL;		//LSB BYTE 2
	bAB1:BOOL;		
	bAB2:BOOL;
	bAB3:BOOL;
	bAB4:BOOL;
	bAB5:BOOL;
	bAB6:BOOL;
	bAB7:BOOL;		//MSB BYTE 2
	bAA0:BOOL;		//LSB BYTE 3
	bAA1:BOOL;
	bAA2:BOOL;
	bAA3:BOOL;
	bAA4:BOOL;
	bAA5:BOOL;
	bAA6:BOOL;
	bAA7:BOOL;		//MSB BYTE 3
END_VAR

VAR_OUTPUT
	dwDW:DWORD;		// Output DWORD
END_VAR

VAR
	PART_BAIXA_BAIXA: BYTE;
	PART_BAIXA_ALTA: BYTE;
	PART_ALTA_BAIXA: BYTE;
	PART_ALTA_ALTA: BYTE;

	WORD_ALTA: WORD;
	WORD_BAIXA: WORD;
END_VAR

PART_BAIXA_BAIXA := PACK(
	B0:= bBB0, 
	B1:= bBB1, 
	B2:= bBB2, 
	B3:= bBB3, 
	B4:= bBB4, 
	B5:= bBB5, 
	B6:= bBB6, 
	B7:= bBB7);
	
PART_BAIXA_ALTA := PACK(
	B0:= bBA0,
	B1:= bBA1, 
	B2:= bBA2, 
	B3:= bBA3, 
	B4:= bBA4, 
	B5:= bBA5, 
	B6:= bBA6, 
	B7:= bBA7);
		
PART_ALTA_BAIXA := PACK(
	B0:= bAB0,
	B1:= bAB1, 
	B2:= bAB2, 
	B3:= bAB3, 
	B4:= bAB4, 
	B5:= bAB5, 
	B6:= bAB6, 
	B7:= bAB7);
	
PART_ALTA_ALTA := PACK(
	B0:= bAA0,
	B1:= bAA1, 
	B2:= bAA2, 
	B3:= bAA3, 
	B4:= bAA4, 
	B5:= bAA5, 
	B6:= bAA6, 
	B7:= bAA7);
	
WORD_BAIXA := BYTE_TO_WORD(PART_BAIXA_BAIXA) OR SHL(BYTE_TO_WORD(PART_BAIXA_ALTA),8); 
WORD_ALTA := BYTE_TO_WORD(PART_ALTA_BAIXA) OR SHL(BYTE_TO_WORD(PART_ALTA_ALTA),8); 
dwDW := WORD_TO_DWORD(WORD_BAIXA) OR SHL(WORD_TO_DWORD(WORD_ALTA),16);

END_FUNCTION_BLOCK

// POUs/PLC/Utils/BitsConversions/Bits_to_word
FUNCTION_BLOCK Bits_to_word
(**********************************************************
Join 16 bits in a WORD Variable  - 29/11/2021
V1.0
*********************************************************)

VAR_INPUT
	bB0:BOOL;		//LSB BYTE 0
	bB1:BOOL;
	bB2:BOOL;
	bB3:BOOL;
	bB4:BOOL;
	bB5:BOOL;
	bB6:BOOL;
	bB7:BOOL;		//MSB BYTE 0
	bA0:BOOL;		//LSB BYTE 1
	bA1:BOOL;
	bA2:BOOL;
	bA3:BOOL;
	bA4:BOOL;
	bA5:BOOL;
	bA6:BOOL;
	bA7:BOOL;		//MSB BYTE 1
END_VAR

VAR_OUTPUT
	wW:WORD;			//WORD Output
END_VAR

VAR
	PARTBAIXA: BYTE;
	PARTALTA: BYTE;
	WORDALTA: WORD;
END_VAR

PARTBAIXA:= PACK(
	B0:= bB0, 
	B1:= bB1, 
	B2:= bB2, 
	B3:= bB3, 
	B4:= bB4, 
	B5:= bB5, 
	B6:= bB6, 
	B7:= bB7);
	
PARTALTA:= PACK(
	B0:= bA0, 
	B1:= bA1, 
	B2:= bA2, 
	B3:= bA3, 
	B4:= bA4, 
	B5:= bA5, 
	B6:= bA6, 
	B7:= bA7);
	
WORDALTA := SHL(BYTE_TO_WORD(PARTALTA),8); 
wW := BYTE_TO_WORD(PARTBAIXA)OR WORDALTA;

END_FUNCTION_BLOCK

// POUs/PLC/Utils/BitsConversions/Dword_to_bits
FUNCTION_BLOCK Dword_to_bits
(**********************************************************
Convert a DWORD variable to 32 bits - 29/11/2021
V1.0 
*********************************************************)

VAR_INPUT
	dwDW:DWORD;		//DWORD Input
END_VAR

VAR_OUTPUT
	bBB0:BOOL;		//LSB BYTE 0
	bBB1:BOOL;
	bBB2:BOOL;
	bBB3:BOOL;
	bBB4:BOOL;
	bBB5:BOOL;
	bBB6:BOOL;
	bBB7:BOOL;		//MSB BYTE 0
	bBA0:BOOL;		//LSB BYTE 1
	bBA1:BOOL;
	bBA2:BOOL;
	bBA3:BOOL;
	bBA4:BOOL;
	bBA5:BOOL;
	bBA6:BOOL;
	bBA7:BOOL;		//MSB BYTE 1
	bAB0:BOOL;		//LSB BYTE 2
	bAB1:BOOL;
	bAB2:BOOL;
	bAB3:BOOL;
	bAB4:BOOL;
	bAB5:BOOL;
	bAB6:BOOL;
	bAB7:BOOL;		//MSB BYTE 2
	bAA0:BOOL;		//LSB BYTE 3
	bAA1:BOOL;
	bAA2:BOOL;
	bAA3:BOOL;
	bAA4:BOOL;
	bAA5:BOOL;
	bAA6:BOOL;
	bAA7:BOOL;		//MSB BYTE 3
END_VAR

VAR

END_VAR



bBB0 := EXTRACT (X:= dwDW, N:=0);
bBB1 := EXTRACT (X:= dwDW, N:=1);
bBB2 := EXTRACT (X:= dwDW, N:=2);
bBB3 := EXTRACT (X:= dwDW, N:=3);
bBB4 := EXTRACT (X:= dwDW, N:=4);
bBB5 := EXTRACT (X:= dwDW, N:=5);
bBB6 := EXTRACT (X:= dwDW, N:=6);
bBB7 := EXTRACT (X:= dwDW, N:=7);
bBA0 := EXTRACT (X:= dwDW, N:=8);
bBA1 := EXTRACT (X:= dwDW, N:=9);
bBA2 := EXTRACT (X:= dwDW, N:=10);
bBA3 := EXTRACT (X:= dwDW, N:=11);
bBA4 := EXTRACT (X:= dwDW, N:=12);
bBA5 := EXTRACT (X:= dwDW, N:=13);
bBA6 := EXTRACT (X:= dwDW, N:=14);
bBA7 := EXTRACT (X:= dwDW, N:=15);
bAB0 := EXTRACT (X:= dwDW, N:=16);
bAB1 := EXTRACT (X:= dwDW, N:=17); 
bAB2 := EXTRACT (X:= dwDW, N:=18);
bAB3 := EXTRACT (X:= dwDW, N:=19);
bAB4 := EXTRACT (X:= dwDW, N:=20);
bAB5 := EXTRACT (X:= dwDW, N:=21);
bAB6 := EXTRACT (X:= dwDW, N:=22);
bAB7 := EXTRACT (X:= dwDW, N:=23);
bAA0 := EXTRACT (X:= dwDW, N:=24);
bAA1 := EXTRACT (X:= dwDW, N:=25);
bAA2 := EXTRACT (X:= dwDW, N:=26);
bAA3 := EXTRACT (X:= dwDW, N:=27);
bAA4 := EXTRACT (X:= dwDW, N:=28);
bAA5 := EXTRACT (X:= dwDW, N:=29);
bAA6 := EXTRACT (X:= dwDW, N:=30);
bAA7 := EXTRACT (X:= dwDW, N:=31);

END_FUNCTION_BLOCK

// POUs/PLC/Utils/BitsConversions/Word_to_bits
FUNCTION_BLOCK word_to_bits
(**********************************************************
Convert a WORD variable to 16 bits - 29/11/2021
V1.0 
*********************************************************)
VAR_INPUT
	wW:WORD;			// WORD Input
END_VAR

VAR_OUTPUT
	bB0:BOOL;		//LSB BYTE 0
	bB1:BOOL;
	bB2:BOOL;
	bB3:BOOL;
	bB4:BOOL;
	bB5:BOOL;
	bB6:BOOL;
	bB7:BOOL;		//MSB BYTE 0
	bA0:BOOL;		//LSB BYTE 1
	bA1:BOOL;
	bA2:BOOL;
	bA3:BOOL;
	bA4:BOOL;
	bA5:BOOL;
	bA6:BOOL;
	bA7:BOOL;		//MSB BYTE 1
END_VAR

VAR

END_VAR

bB0 := EXTRACT (X:= wW, N:=0);
bB1 := EXTRACT (X:= wW, N:=1);
bB2 := EXTRACT (X:= wW, N:=2);
bB3 := EXTRACT (X:= wW, N:=3);
bB4 := EXTRACT (X:= wW, N:=4);
bB5 := EXTRACT (X:= wW, N:=5);
bB6 := EXTRACT (X:= wW, N:=6);
bB7 := EXTRACT (X:= wW, N:=7);
bA0 := EXTRACT (X:= wW, N:=8);
bA1 := EXTRACT (X:= wW, N:=9);
bA2 := EXTRACT (X:= wW, N:=10);
bA3 := EXTRACT (X:= wW, N:=11);
bA4 := EXTRACT (X:= wW, N:=12);
bA5 := EXTRACT (X:= wW, N:=13);
bA6 := EXTRACT (X:= wW, N:=14);
bA7 := EXTRACT (X:= wW, N:=15);

END_FUNCTION_BLOCK

// POUs/PLC/Utils/Counters/Calcul_Frequencia
FUNCTION_BLOCK Calcul_Frequencia
(**********************************************************
Calculate an counter frequency - 26/11/2021
V1.00
*********************************************************)
VAR_INPUT
	xStart:BOOL; 		// Start executing the function
	rCounter:REAL;		// Input of the counter value
END_VAR

VAR_OUTPUT
	rFrequency_REAL:REAL;		//Frequency Output (REAL)
	dwFrequency_DWORD:DWORD;		//Frequency Output (DWORD)
END_VAR

VAR
	TempoContador: TON;
	tempsConta: TIME;
	div2: REAL;
	zr: BOOL;
	cum: REAL;
	adiv: REAL;
	hz: REAL;
END_VAR

TempoContador(IN:=xStart , PT:=T#7D, Q=> , ET=>tempsConta);

div2 := TIME_TO_REAL(tempsConta);

IF	div2 = 0 
	THEN
		zr := TRUE;
	ELSE
		zr := FALSE;
END_IF

IF zr 
	THEN
		cum := RCounter;
END_IF

adiv := (RCounter - cum);

IF NOT zr 
	THEN
		hz := (1000*(adiv/div2));
	ELSE
		hz := 0;
END_IF

rFrequency_REAL := hz;
dwFrequency_DWORD := REAL_TO_DWORD(hz);

END_FUNCTION_BLOCK

// POUs/PLC/Utils/FreqCycle/CalcFreq
FUNCTION_BLOCK CalcFreq
(**********************************************************
 - 29/11/2021
V1.00
*********************************************************)

VAR_INPUT

END_VAR

VAR_OUTPUT
	wFreq:WORD;			//Frrequency Output
END_VAR

VAR
	tempor1:TON;
	pols: BOOL;
	c: WORD;
	b: WORD;
END_VAR

tempor1 (in:=NOT(tempor1.Q), PT:=t#1s, Q=>pols);

IF pols=TRUE
	THEN
	c:=a-b;
	IF a>=9999
		THEN
		a:=0;
	END_IF
	b:=a;
END_IF

wFreq:=C;

END_FUNCTION_BLOCK

// POUs/PLC/Utils/Timers/fBPulse1s
FUNCTION_BLOCK fBPulse1s
VAR_OUTPUT
	xFlanco: BOOL;
	xOut: BOOL;
END_VAR
VAR
	tTempo: Ton;
	iSeg: UDINT;
	pPulse: R_trig;
	iSeg_Ant: UDINT;
	PULSO: BLINK;
END_VAR



tTempo(IN:=NOT(tTempo.Q) , PT:=T#7D );
iSeg:=TIME_TO_DWORD(tTempo.ET)/1000;
pPulse(CLK:= (iSeg>iSeg_Ant) );
iSeg_Ant:=iSeg;

xFlanco:=pPulse.Q;

PULSO(ENABLE:= TRUE, TIMELOW:= T#1S, TIMEHIGH:= T#1S, OUT=> xOut);

END_FUNCTION_BLOCK
